SPLINE
SPL {X  -154.923, Y  +342.556, Z    +0.000, E1   +23.930, E3 +323700.309}
SPL {X  -158.138, Y  +358.230, Z    +0.000, E1   +16.243, E3 +323709.267}
SPL {X  -159.407, Y  +368.849, Z    +0.000, E1   +10.504, E3 +323712.867}
SPL {X  -159.931, Y  +378.162, Z    +0.000, E1    +5.020, E3 +323714.852}
SPL {X  -159.990, Y  +384.616, Z    +0.000, E1    +0.627, E3 +323715.691}
SPL {X  -159.990, Y  +387.962, Z    +0.000, E1    -2.241, E3 +323716.048}
SPL {X  -159.990, Y  +390.921, Z    +0.000, E1    -5.111, E3 +323716.413}
SPL {X  -159.990, Y  +395.719, Z    +0.000, E1   -10.396, E3 +323717.232}
SPL {X  -159.990, Y  +400.739, Z    +0.000, E1   -16.236, E3 +323718.430}
SPL {X  -159.990, Y  +409.482, Z    +0.000, E1   -25.418, E3 +323721.635}
SPL {X  -159.990, Y  +440.741, Z    +0.000, E1   -43.570, E3 +323742.292}
SPL {X  -159.990, Y  +488.072, Z    +0.000, E1   -48.834, E3 +323803.414}
SPL {X  -159.990, Y  +495.397, Z    +0.000, E1   -48.860, E3 +323816.963}
SPL {X  -159.990, Y  +502.531, Z    +0.000, E1   -48.834, E3 +323830.242}
SPL {X  -159.990, Y  +508.013, Z    +0.000, E1   -48.835, E3 +323840.377}
SPL {X  -159.990, Y  +513.813, Z    +0.000, E1   -48.843, E3 +323851.125}
SPL {X  -159.990, Y  +522.177, Z    +0.000, E1   -48.881, E3 +323866.602}
SPL {X  -159.990, Y  +532.076, Z    +0.000, E1   -48.872, E3 +323884.975}
SPL {X  -159.990, Y  +539.248, Z    +0.000, E1   -48.832, E3 +323898.343}
SPL {X  -159.990, Y  +544.926, Z    +0.000, E1   -48.835, E3 +323908.872}
SPL {X  -159.990, Y  +550.252, Z    +0.000, E1   -48.827, E3 +323918.778}
SPL {X  -159.990, Y  +555.692, Z    +0.000, E1   -48.830, E3 +323928.875}
SPL {X  -159.990, Y  +561.308, Z    +0.000, E1   -48.827, E3 +323939.322}
SPL {X  -159.990, Y  +566.669, Z    +0.000, E1   -48.820, E3 +323949.271}
SPL {X  -159.990, Y  +572.248, Z    +0.000, E1   -48.830, E3 +323959.616}
SPL {X  -159.990, Y  +577.770, Z    +0.000, E1   -48.821, E3 +323969.863}
SPL {X  -159.990, Y  +583.108, Z    +0.000, E1   -48.828, E3 +323979.765}
SPL {X  -159.990, Y  +588.804, Z    +0.000, E1   -48.829, E3 +323990.322}
SPL {X  -159.990, Y  +594.280, Z    +0.000, E1   -48.826, E3 +324000.484}
SPL {X  -159.990, Y  +600.107, Z    +0.000, E1   -48.833, E3 +324011.298}
SPL {X  -159.990, Y  +605.910, Z    +0.000, E1   -48.823, E3 +324022.077}
SPL {X  -159.990, Y  +611.566, Z    +0.000, E1   -48.829, E3 +324032.566}
SPL {X  -159.990, Y  +617.357, Z    +0.000, E1   -48.824, E3 +324043.321}
SPL {X  -159.990, Y  +622.965, Z    +0.000, E1   -48.826, E3 +324053.720}
SPL {X  -159.990, Y  +629.255, Z    +0.000, E1   -48.834, E3 +324065.387}
SPL {X  -159.990, Y  +634.905, Z    +0.000, E1   -48.821, E3 +324075.884}
SPL {X  -159.990, Y  +640.372, Z    +0.000, E1   -48.828, E3 +324086.021}
SPL {X  -159.990, Y  +646.939, Z    +0.000, E1   -48.838, E3 +324098.191}
SPL {X  -159.990, Y  +653.448, Z    +0.000, E1   -48.827, E3 +324110.286}
SPL {X  -159.990, Y  +659.039, Z    +0.000, E1   -48.826, E3 +324120.650}
SPL {X  -159.990, Y  +664.817, Z    +0.000, E1   -48.832, E3 +324131.365}
SPL {X  -159.990, Y  +671.221, Z    +0.000, E1   -48.836, E3 +324143.238}
SPL {X  -159.887, Y  +677.230, Z    +0.000, E1   -48.811, E3 +324154.504}
SPL {X  -159.602, Y  +682.629, Z    +0.000, E1   -48.761, E3 +324164.837}
SPL {X  -159.150, Y  +687.876, Z    +0.000, E1   -48.673, E3 +324175.076}
SPL {X  -158.569, Y  +692.776, Z    +0.000, E1   -48.570, E3 +324184.784}
SPL {X  -157.870, Y  +697.458, Z    +0.000, E1   -48.439, E3 +324194.213}
SPL {X  -157.028, Y  +702.144, Z    +0.000, E1   -48.297, E3 +324203.761}
SPL {X  -155.977, Y  +707.110, Z    +0.000, E1   -48.106, E3 +324214.065}
SPL {X  -154.657, Y  +712.464, Z    +0.000, E1   -47.874, E3 +324225.349}
SPL {X  -153.406, Y  +716.924, Z    +0.000, E1   -47.628, E3 +324234.915}
SPL {X  -152.020, Y  +721.367, Z    +0.000, E1   -47.374, E3 +324244.566}
SPL {X  -150.440, Y  +725.947, Z    +0.000, E1   -47.070, E3 +324254.671}
SPL {X  -148.730, Y  +730.459, Z    +0.000, E1   -46.749, E3 +324264.722}
SPL {X  -147.178, Y  +734.233, Z    +0.000, E1   -46.439, E3 +324273.256}
SPL {X  -140.263, Y  +748.461, Z    +0.000, E1   -42.675, E3 +324331.594}
ENDSPLINE

SPLINE
SPL {X  -141.835, Y  +745.525, Z    +0.000, E1   -39.068, E3 +324363.595}
SPL {X  -152.406, Y  +720.176, Z    +0.000, E1   -27.814, E3 +324414.808}
SPL {X  -158.165, Y  +695.595, Z    +0.000, E1   -16.189, E3 +324430.706}
SPL {X  -159.572, Y  +683.063, Z    +0.000, E1    -9.282, E3 +324434.713}
SPL {X  -159.928, Y  +675.946, Z    +0.000, E1    -5.007, E3 +324436.134}
SPL {X  -159.990, Y  +671.468, Z    +0.000, E1    -2.030, E3 +324436.730}
SPL {X  -159.990, Y  +667.678, Z    +0.000, E1    +0.783, E3 +324437.080}
SPL {X  -159.990, Y  +663.139, Z    +0.000, E1    +5.135, E3 +324437.597}
SPL {X  -159.990, Y  +658.551, Z    +0.000, E1   +10.313, E3 +324438.371}
SPL {X  -159.990, Y  +653.526, Z    +0.000, E1   +16.156, E3 +324439.606}
SPL {X  -159.990, Y  +644.434, Z    +0.000, E1   +25.921, E3 +324442.801}
SPL {X  -159.990, Y  +612.255, Z    +0.000, E1   +44.102, E3 +324464.682}
SPL {X  -159.990, Y  +562.879, Z    +0.000, E1   +49.634, E3 +324526.271}
SPL {X  -159.990, Y  +554.544, Z    +0.000, E1   +49.649, E3 +324541.296}
SPL {X  -159.990, Y  +547.278, Z    +0.000, E1   +49.619, E3 +324554.455}
SPL {X  -159.990, Y  +540.489, Z    +0.000, E1   +49.634, E3 +324566.681}
SPL {X  -159.990, Y  +530.983, Z    +0.000, E1   +49.676, E3 +324583.752}
SPL {X  -159.990, Y  +522.804, Z    +0.000, E1   +49.620, E3 +324598.592}
SPL {X  -159.990, Y  +515.173, Z    +0.000, E1   +49.653, E3 +324612.330}
SPL {X  -159.990, Y  +505.472, Z    +0.000, E1   +49.465, E3 +324631.135}
ENDSPLINE

SPLINE
SPL {X  -159.990, Y  +518.841, Z    +0.000, E1   +41.643, E3 +324649.543}
ENDSPLINE

SPLINE
SPL {X  -159.990, Y  +508.096, Z    +0.000, E1   +42.952, E3 +324666.810}
SPL {X  -159.990, Y  +500.642, Z    +0.000, E1   +43.747, E3 +324678.731}
SPL {X  -159.990, Y  +495.820, Z    +0.000, E1   +44.207, E3 +324686.618}
SPL {X  -159.990, Y  +487.435, Z    +0.000, E1   +45.185, E3 +324698.910}
SPL {X  -159.990, Y  +477.648, Z    +0.000, E1   +46.080, E3 +324713.907}
SPL {X  -159.990, Y  +469.952, Z    +0.000, E1   +46.750, E3 +324725.415}
SPL {X  -159.990, Y  +460.762, Z    +0.000, E1   +47.755, E3 +324737.551}
SPL {X  -159.990, Y  +451.028, Z    +0.000, E1   +48.723, E3 +324750.163}
SPL {X  -159.990, Y  +441.023, Z    +0.000, E1   +49.655, E3 +324762.997}
SPL {X  -159.990, Y  +431.096, Z    +0.000, E1   +50.075, E3 +324778.285}
SPL {X  -159.990, Y  +423.834, Z    +0.000, E1   +50.037, E3 +324791.258}
SPL {X  -159.990, Y  +417.693, Z    +0.000, E1   +50.049, E3 +324802.156}
SPL {X  -159.990, Y  +411.447, Z    +0.000, E1   +50.039, E3 +324813.275}
SPL {X  -159.990, Y  +406.170, Z    +0.000, E1   +50.036, E3 +324822.647}
SPL {X  -159.990, Y  +399.787, Z    +0.000, E1   +50.064, E3 +324833.955}
SPL {X  -159.990, Y  +393.038, Z    +0.000, E1   +50.038, E3 +324845.989}
SPL {X  -159.990, Y  +387.356, Z    +0.000, E1   +50.042, E3 +324856.100}
SPL {X  -159.956, Y  +379.183, Z    +0.000, E1   +50.071, E3 +324870.614}
SPL {X  -159.413, Y  +368.921, Z    +0.000, E1   +49.998, E3 +324889.389}
SPL {X  -158.412, Y  +360.086, Z    +0.000, E1   +49.787, E3 +324906.191}
SPL {X  -157.077, Y  +352.107, Z    +0.000, E1   +49.567, E3 +324921.742}
SPL {X  -155.744, Y  +345.884, Z    +0.000, E1   +49.283, E3 +324934.229}
SPL {X  -154.686, Y  +341.646, Z    +0.000, E1   +49.094, E3 +324942.855}
SPL {X  -153.089, Y  +336.017, Z    +0.000, E1   +48.817, E3 +324954.464}
SPL {X  -151.481, Y  +331.019, Z    +0.000, E1   +48.491, E3 +324965.012}
SPL {X  -149.787, Y  +326.281, Z    +0.000, E1   +48.192, E3 +324975.100}
SPL {X  -148.124, Y  +322.035, Z    +0.000, E1   +47.846, E3 +324984.324}
SPL {X  -146.510, Y  +318.222, Z    +0.000, E1   +47.558, E3 +324992.636}
SPL {X  -141.189, Y  +307.250, Z    +0.000, E1   +40.067, E3 +325078.810}
ENDSPLINE

SPLINE
SPL {X  -154.923, Y  +342.556, Z    +0.000, E1   +23.930, E3 +325140.309}
SPL {X  -158.138, Y  +358.230, Z    +0.000, E1   +16.243, E3 +325149.267}
SPL {X  -159.647, Y  +372.034, Z    +0.000, E1    +8.739, E3 +325153.631}
SPL {X  -159.989, Y  +381.927, Z    +0.000, E1    +2.565, E3 +325155.391}
SPL {X  -159.990, Y  +386.909, Z    +0.000, E1    -1.211, E3 +325155.934}
SPL {X  -159.990, Y  +390.921, Z    +0.000, E1    -5.111, E3 +325156.413}
SPL {X  -159.990, Y  +395.719, Z    +0.000, E1   -10.396, E3 +325157.232}
SPL {X  -159.990, Y  +400.739, Z    +0.000, E1   -16.236, E3 +325158.430}
SPL {X  -159.990, Y  +409.482, Z    +0.000, E1   -25.418, E3 +325161.635}
SPL {X  -159.990, Y  +440.741, Z    +0.000, E1   -43.570, E3 +325182.292}
SPL {X  -159.990, Y  +488.072, Z    +0.000, E1   -48.834, E3 +325243.414}
SPL {X  -159.990, Y  +495.397, Z    +0.000, E1   -48.860, E3 +325256.963}
SPL {X  -159.990, Y  +502.531, Z    +0.000, E1   -48.834, E3 +325270.242}
SPL {X  -159.990, Y  +508.013, Z    +0.000, E1   -48.835, E3 +325280.377}
SPL {X  -159.990, Y  +513.813, Z    +0.000, E1   -48.843, E3 +325291.125}
SPL {X  -159.990, Y  +519.614, Z    +0.000, E1   -48.832, E3 +325301.926}
SPL {X  -159.990, Y  +527.523, Z    +0.000, E1   -48.881, E3 +325316.507}
SPL {X  -159.990, Y  +537.185, Z    +0.000, E1   -48.874, E3 +325334.454}
SPL {X  -159.990, Y  +544.926, Z    +0.000, E1   -48.835, E3 +325348.872}
SPL {X  -159.990, Y  +550.252, Z    +0.000, E1   -48.827, E3 +325358.778}
SPL {X  -159.990, Y  +555.692, Z    +0.000, E1   -48.830, E3 +325368.875}
SPL {X  -159.990, Y  +561.308, Z    +0.000, E1   -48.827, E3 +325379.322}
SPL {X  -159.990, Y  +566.669, Z    +0.000, E1   -48.820, E3 +325389.271}
SPL {X  -159.990, Y  +572.248, Z    +0.000, E1   -48.830, E3 +325399.616}
SPL {X  -159.990, Y  +577.770, Z    +0.000, E1   -48.821, E3 +325409.863}
SPL {X  -159.990, Y  +583.108, Z    +0.000, E1   -48.828, E3 +325419.765}
SPL {X  -159.990, Y  +588.804, Z    +0.000, E1   -48.829, E3 +325430.322}
SPL {X  -159.990, Y  +594.280, Z    +0.000, E1   -48.826, E3 +325440.484}
SPL {X  -159.990, Y  +600.107, Z    +0.000, E1   -48.833, E3 +325451.298}
SPL {X  -159.990, Y  +605.910, Z    +0.000, E1   -48.823, E3 +325462.077}
SPL {X  -159.990, Y  +611.566, Z    +0.000, E1   -48.829, E3 +325472.566}
SPL {X  -159.990, Y  +617.357, Z    +0.000, E1   -48.824, E3 +325483.321}
SPL {X  -159.990, Y  +622.965, Z    +0.000, E1   -48.826, E3 +325493.720}
SPL {X  -159.990, Y  +629.255, Z    +0.000, E1   -48.834, E3 +325505.387}
SPL {X  -159.990, Y  +634.905, Z    +0.000, E1   -48.821, E3 +325515.884}
SPL {X  -159.990, Y  +640.372, Z    +0.000, E1   -48.828, E3 +325526.021}
SPL {X  -159.990, Y  +646.939, Z    +0.000, E1   -48.838, E3 +325538.191}
SPL {X  -159.990, Y  +653.448, Z    +0.000, E1   -48.827, E3 +325550.286}
SPL {X  -159.990, Y  +659.039, Z    +0.000, E1   -48.826, E3 +325560.650}
SPL {X  -159.990, Y  +664.817, Z    +0.000, E1   -48.832, E3 +325571.365}
SPL {X  -159.990, Y  +671.221, Z    +0.000, E1   -48.836, E3 +325583.238}
SPL {X  -159.887, Y  +677.230, Z    +0.000, E1   -48.811, E3 +325594.504}
SPL {X  -159.602, Y  +682.629, Z    +0.000, E1   -48.761, E3 +325604.837}
SPL {X  -159.150, Y  +687.876, Z    +0.000, E1   -48.673, E3 +325615.076}
SPL {X  -158.569, Y  +692.776, Z    +0.000, E1   -48.570, E3 +325624.784}
SPL {X  -157.870, Y  +697.458, Z    +0.000, E1   -48.439, E3 +325634.213}
SPL {X  -157.028, Y  +702.144, Z    +0.000, E1   -48.297, E3 +325643.761}
SPL {X  -155.977, Y  +707.110, Z    +0.000, E1   -48.106, E3 +325654.065}
SPL {X  -154.657, Y  +712.464, Z    +0.000, E1   -47.874, E3 +325665.349}
SPL {X  -153.406, Y  +716.924, Z    +0.000, E1   -47.628, E3 +325674.915}
SPL {X  -152.020, Y  +721.367, Z    +0.000, E1   -47.374, E3 +325684.566}
SPL {X  -150.440, Y  +725.947, Z    +0.000, E1   -47.070, E3 +325694.671}
SPL {X  -148.730, Y  +730.459, Z    +0.000, E1   -46.749, E3 +325704.722}
SPL {X  -147.178, Y  +734.233, Z    +0.000, E1   -46.439, E3 +325713.256}
SPL {X  -140.263, Y  +748.461, Z    +0.000, E1   -42.675, E3 +325771.594}
ENDSPLINE

SPLINE
SPL {X  -141.835, Y  +745.525, Z    +0.000, E1   -39.068, E3 +325803.595}
SPL {X  -152.406, Y  +720.176, Z    +0.000, E1   -27.814, E3 +325854.808}
SPL {X  -158.165, Y  +695.595, Z    +0.000, E1   -16.189, E3 +325870.706}
SPL {X  -159.572, Y  +683.063, Z    +0.000, E1    -9.282, E3 +325874.713}
SPL {X  -159.928, Y  +675.946, Z    +0.000, E1    -5.007, E3 +325876.134}
SPL {X  -159.990, Y  +671.468, Z    +0.000, E1    -2.030, E3 +325876.730}
SPL {X  -159.990, Y  +667.678, Z    +0.000, E1    +0.783, E3 +325877.080}
SPL {X  -159.990, Y  +663.139, Z    +0.000, E1    +5.135, E3 +325877.597}
SPL {X  -159.990, Y  +658.551, Z    +0.000, E1   +10.313, E3 +325878.371}
SPL {X  -159.990, Y  +653.526, Z    +0.000, E1   +16.156, E3 +325879.606}
SPL {X  -159.990, Y  +644.434, Z    +0.000, E1   +25.921, E3 +325882.801}
SPL {X  -159.990, Y  +612.255, Z    +0.000, E1   +44.102, E3 +325904.682}
SPL {X  -159.990, Y  +562.879, Z    +0.000, E1   +49.634, E3 +325966.271}
SPL {X  -159.990, Y  +554.544, Z    +0.000, E1   +49.649, E3 +325981.296}
SPL {X  -159.990, Y  +547.278, Z    +0.000, E1   +49.619, E3 +325994.455}
SPL {X  -159.990, Y  +540.489, Z    +0.000, E1   +49.634, E3 +326006.681}
SPL {X  -159.990, Y  +530.983, Z    +0.000, E1   +49.676, E3 +326023.752}
SPL {X  -159.990, Y  +522.804, Z    +0.000, E1   +49.620, E3 +326038.592}
SPL {X  -159.990, Y  +515.173, Z    +0.000, E1   +49.653, E3 +326052.330}
SPL {X  -159.990, Y  +505.472, Z    +0.000, E1   +49.465, E3 +326071.135}
ENDSPLINE

SPLINE
SPL {X  -159.990, Y  +520.622, Z    +0.000, E1   +41.395, E3 +326086.672}
ENDSPLINE

SPLINE
SPL {X  -159.990, Y  +512.735, Z    +0.000, E1   +42.369, E3 +326099.523}
SPL {X  -159.990, Y  +505.924, Z    +0.000, E1   +43.199, E3 +326110.181}
SPL {X  -159.990, Y  +497.983, Z    +0.000, E1   +44.027, E3 +326123.054}
SPL {X  -159.990, Y  +489.703, Z    +0.000, E1   +44.938, E3 +326135.473}
SPL {X  -159.990, Y  +482.131, Z    +0.000, E1   +45.680, E3 +326147.053}
SPL {X  -159.990, Y  +472.111, Z    +0.000, E1   +46.581, E3 +326162.185}
SPL {X  -159.990, Y  +462.892, Z    +0.000, E1   +47.497, E3 +326174.899}
SPL {X  -159.990, Y  +450.424, Z    +0.000, E1   +48.824, E3 +326190.863}
SPL {X  -159.990, Y  +436.919, Z    +0.000, E1   +49.944, E3 +326208.632}
SPL {X  -159.990, Y  +429.517, Z    +0.000, E1   +50.043, E3 +326221.146}
SPL {X  -159.990, Y  +423.834, Z    +0.000, E1   +50.037, E3 +326231.258}
SPL {X  -159.990, Y  +417.693, Z    +0.000, E1   +50.049, E3 +326242.156}
SPL {X  -159.990, Y  +411.447, Z    +0.000, E1   +50.039, E3 +326253.275}
SPL {X  -159.990, Y  +403.654, Z    +0.000, E1   +50.076, E3 +326267.065}
SPL {X  -159.990, Y  +394.612, Z    +0.000, E1   +50.064, E3 +326283.153}
SPL {X  -159.990, Y  +387.356, Z    +0.000, E1   +50.042, E3 +326296.100}
SPL {X  -159.956, Y  +379.183, Z    +0.000, E1   +50.071, E3 +326310.614}
SPL {X  -159.413, Y  +368.921, Z    +0.000, E1   +49.998, E3 +326329.389}
SPL {X  -158.412, Y  +360.086, Z    +0.000, E1   +49.787, E3 +326346.191}
SPL {X  -157.077, Y  +352.107, Z    +0.000, E1   +49.567, E3 +326361.742}
SPL {X  -155.744, Y  +345.884, Z    +0.000, E1   +49.283, E3 +326374.229}
SPL {X  -154.686, Y  +341.646, Z    +0.000, E1   +49.094, E3 +326382.855}
SPL {X  -153.089, Y  +336.017, Z    +0.000, E1   +48.817, E3 +326394.464}
SPL {X  -151.481, Y  +331.019, Z    +0.000, E1   +48.491, E3 +326405.012}
SPL {X  -150.221, Y  +327.451, Z    +0.000, E1   +48.251, E3 +326412.616}
SPL {X  -148.587, Y  +323.181, Z    +0.000, E1   +47.960, E3 +326421.800}
SPL {X  -146.510, Y  +318.222, Z    +0.000, E1   +47.558, E3 +326432.636}
SPL {X  -141.189, Y  +307.250, Z    +0.000, E1   +40.067, E3 +326518.810}
ENDSPLINE

SPLINE
SPL {X  -154.923, Y  +342.556, Z    +0.000, E1   +23.930, E3 +326580.309}
SPL {X  -158.138, Y  +358.230, Z    +0.000, E1   +16.243, E3 +326589.267}
SPL {X  -159.407, Y  +368.849, Z    +0.000, E1   +10.504, E3 +326592.867}
SPL {X  -159.931, Y  +378.162, Z    +0.000, E1    +5.020, E3 +326594.852}
SPL {X  -159.990, Y  +383.297, Z    +0.000, E1    +1.526, E3 +326595.557}
SPL {X  -159.990, Y  +386.909, Z    +0.000, E1    -1.211, E3 +326595.934}
SPL {X  -159.990, Y  +390.921, Z    +0.000, E1    -5.111, E3 +326596.413}
SPL {X  -159.990, Y  +395.719, Z    +0.000, E1   -10.396, E3 +326597.232}
SPL {X  -159.990, Y  +400.739, Z    +0.000, E1   -16.236, E3 +326598.430}
SPL {X  -159.990, Y  +407.669, Z    +0.000, E1   -23.731, E3 +326600.753}
SPL {X  -159.990, Y  +417.102, Z    +0.000, E1   -32.094, E3 +326605.313}
SPL {X  -159.990, Y  +440.741, Z    +0.000, E1   -43.570, E3 +326622.292}
SPL {X  -159.990, Y  +488.072, Z    +0.000, E1   -48.834, E3 +326683.414}
SPL {X  -159.990, Y  +495.397, Z    +0.000, E1   -48.860, E3 +326696.963}
SPL {X  -159.990, Y  +502.531, Z    +0.000, E1   -48.834, E3 +326710.242}
SPL {X  -159.990, Y  +508.013, Z    +0.000, E1   -48.835, E3 +326720.377}
SPL {X  -159.990, Y  +513.813, Z    +0.000, E1   -48.843, E3 +326731.125}
SPL {X  -159.990, Y  +522.177, Z    +0.000, E1   -48.881, E3 +326746.602}
SPL {X  -159.990, Y  +532.076, Z    +0.000, E1   -48.872, E3 +326764.975}
SPL {X  -159.990, Y  +539.248, Z    +0.000, E1   -48.832, E3 +326778.343}
SPL {X  -159.990, Y  +544.926, Z    +0.000, E1   -48.835, E3 +326788.872}
SPL {X  -159.990, Y  +550.252, Z    +0.000, E1   -48.827, E3 +326798.778}
SPL {X  -159.990, Y  +555.692, Z    +0.000, E1   -48.830, E3 +326808.875}
SPL {X  -159.990, Y  +561.308, Z    +0.000, E1   -48.827, E3 +326819.322}
SPL {X  -159.990, Y  +566.669, Z    +0.000, E1   -48.820, E3 +326829.271}
SPL {X  -159.990, Y  +572.248, Z    +0.000, E1   -48.830, E3 +326839.616}
SPL {X  -159.990, Y  +577.770, Z    +0.000, E1   -48.821, E3 +326849.863}
SPL {X  -159.990, Y  +583.108, Z    +0.000, E1   -48.828, E3 +326859.765}
SPL {X  -159.990, Y  +588.804, Z    +0.000, E1   -48.829, E3 +326870.322}
SPL {X  -159.990, Y  +594.280, Z    +0.000, E1   -48.826, E3 +326880.484}
SPL {X  -159.990, Y  +600.107, Z    +0.000, E1   -48.833, E3 +326891.298}
SPL {X  -159.990, Y  +605.910, Z    +0.000, E1   -48.823, E3 +326902.077}
SPL {X  -159.990, Y  +611.566, Z    +0.000, E1   -48.829, E3 +326912.566}
SPL {X  -159.990, Y  +617.357, Z    +0.000, E1   -48.824, E3 +326923.321}
SPL {X  -159.990, Y  +622.965, Z    +0.000, E1   -48.826, E3 +326933.720}
SPL {X  -159.990, Y  +629.255, Z    +0.000, E1   -48.834, E3 +326945.387}
SPL {X  -159.990, Y  +634.905, Z    +0.000, E1   -48.821, E3 +326955.884}
SPL {X  -159.990, Y  +640.372, Z    +0.000, E1   -48.828, E3 +326966.021}
SPL {X  -159.990, Y  +646.939, Z    +0.000, E1   -48.838, E3 +326978.191}
SPL {X  -159.990, Y  +653.448, Z    +0.000, E1   -48.827, E3 +326990.286}
SPL {X  -159.990, Y  +659.039, Z    +0.000, E1   -48.826, E3 +327000.650}
SPL {X  -159.990, Y  +664.817, Z    +0.000, E1   -48.832, E3 +327011.365}
SPL {X  -159.990, Y  +671.221, Z    +0.000, E1   -48.836, E3 +327023.238}
SPL {X  -159.887, Y  +677.230, Z    +0.000, E1   -48.811, E3 +327034.504}
SPL {X  -159.602, Y  +682.629, Z    +0.000, E1   -48.761, E3 +327044.837}
SPL {X  -159.150, Y  +687.876, Z    +0.000, E1   -48.673, E3 +327055.076}
SPL {X  -158.569, Y  +692.776, Z    +0.000, E1   -48.570, E3 +327064.784}
SPL {X  -157.870, Y  +697.458, Z    +0.000, E1   -48.439, E3 +327074.213}
SPL {X  -157.028, Y  +702.144, Z    +0.000, E1   -48.297, E3 +327083.761}
SPL {X  -155.977, Y  +707.110, Z    +0.000, E1   -48.106, E3 +327094.065}
SPL {X  -154.657, Y  +712.464, Z    +0.000, E1   -47.874, E3 +327105.349}
SPL {X  -153.406, Y  +716.924, Z    +0.000, E1   -47.628, E3 +327114.915}
SPL {X  -152.020, Y  +721.367, Z    +0.000, E1   -47.374, E3 +327124.566}
SPL {X  -150.440, Y  +725.947, Z    +0.000, E1   -47.070, E3 +327134.671}
SPL {X  -148.730, Y  +730.459, Z    +0.000, E1   -46.749, E3 +327144.722}
SPL {X  -147.178, Y  +734.233, Z    +0.000, E1   -46.439, E3 +327153.256}
SPL {X  -140.263, Y  +748.461, Z    +0.000, E1   -42.675, E3 +327211.594}
ENDSPLINE

SPLINE
SPL {X  -141.835, Y  +745.525, Z    +0.000, E1   -39.068, E3 +327243.595}
SPL {X  -152.406, Y  +720.176, Z    +0.000, E1   -27.814, E3 +327294.808}
SPL {X  -157.542, Y  +699.382, Z    +0.000, E1   -18.086, E3 +327309.141}
SPL {X  -159.386, Y  +685.393, Z    +0.000, E1   -10.664, E3 +327314.095}
SPL {X  -159.928, Y  +675.946, Z    +0.000, E1    -5.007, E3 +327316.134}
SPL {X  -159.990, Y  +671.468, Z    +0.000, E1    -2.030, E3 +327316.730}
SPL {X  -159.990, Y  +667.678, Z    +0.000, E1    +0.783, E3 +327317.080}
SPL {X  -159.990, Y  +663.139, Z    +0.000, E1    +5.135, E3 +327317.597}
SPL {X  -159.990, Y  +658.551, Z    +0.000, E1   +10.313, E3 +327318.371}
SPL {X  -159.990, Y  +653.526, Z    +0.000, E1   +16.156, E3 +327319.606}
SPL {X  -159.990, Y  +644.434, Z    +0.000, E1   +25.921, E3 +327322.801}
SPL {X  -159.990, Y  +612.255, Z    +0.000, E1   +44.102, E3 +327344.682}
SPL {X  -159.990, Y  +561.053, Z    +0.000, E1   +49.668, E3 +327409.515}
SPL {X  -159.990, Y  +552.984, Z    +0.000, E1   +49.619, E3 +327424.156}
SPL {X  -159.990, Y  +547.278, Z    +0.000, E1   +49.619, E3 +327434.455}
SPL {X  -159.990, Y  +538.738, Z    +0.000, E1   +49.672, E3 +327449.779}
SPL {X  -159.990, Y  +529.436, Z    +0.000, E1   +49.638, E3 +327466.603}
SPL {X  -159.990, Y  +520.280, Z    +0.000, E1   +49.665, E3 +327483.082}
SPL {X  -159.990, Y  +511.038, Z    +0.000, E1   +49.636, E3 +327499.832}
SPL {X  -159.990, Y  +504.260, Z    +0.000, E1   +49.614, E3 +327512.105}
SPL {X  -159.990, Y  +503.881, Z    +0.000, E1   +48.376, E3 +327520.092}
ENDSPLINE

SPLINE
SPL {X  -159.990, Y  +520.622, Z    +0.000, E1   +41.395, E3 +327526.672}
ENDSPLINE

SPLINE
SPL {X  -159.990, Y  +512.735, Z    +0.000, E1   +42.369, E3 +327539.523}
SPL {X  -159.990, Y  +505.924, Z    +0.000, E1   +43.199, E3 +327550.181}
SPL {X  -159.990, Y  +497.983, Z    +0.000, E1   +44.027, E3 +327563.054}
SPL {X  -159.990, Y  +489.703, Z    +0.000, E1   +44.938, E3 +327575.473}
SPL {X  -159.990, Y  +484.712, Z    +0.000, E1   +45.426, E3 +327583.087}
SPL {X  -159.990, Y  +477.648, Z    +0.000, E1   +46.080, E3 +327593.907}
SPL {X  -159.990, Y  +469.952, Z    +0.000, E1   +46.750, E3 +327605.415}
SPL {X  -159.990, Y  +462.892, Z    +0.000, E1   +47.497, E3 +327614.899}
SPL {X  -159.990, Y  +450.424, Z    +0.000, E1   +48.824, E3 +327630.863}
SPL {X  -159.990, Y  +436.919, Z    +0.000, E1   +49.944, E3 +327648.632}
SPL {X  -159.990, Y  +429.517, Z    +0.000, E1   +50.043, E3 +327661.146}
SPL {X  -159.990, Y  +423.834, Z    +0.000, E1   +50.037, E3 +327671.258}
SPL {X  -159.990, Y  +417.693, Z    +0.000, E1   +50.049, E3 +327682.156}
SPL {X  -159.990, Y  +408.922, Z    +0.000, E1   +50.085, E3 +327697.686}
SPL {X  -159.990, Y  +399.787, Z    +0.000, E1   +50.064, E3 +327713.955}
SPL {X  -159.990, Y  +393.038, Z    +0.000, E1   +50.038, E3 +327725.989}
SPL {X  -159.990, Y  +385.182, Z    +0.000, E1   +50.081, E3 +327739.906}
SPL {X  -159.906, Y  +377.302, Z    +0.000, E1   +50.024, E3 +327754.067}
SPL {X  -159.545, Y  +370.569, Z    +0.000, E1   +49.982, E3 +327766.380}
SPL {X  -158.871, Y  +363.614, Z    +0.000, E1   +49.855, E3 +327779.459}
SPL {X  -158.179, Y  +358.495, Z    +0.000, E1   +49.715, E3 +327789.308}
SPL {X  -157.354, Y  +353.576, Z    +0.000, E1   +49.583, E3 +327798.894}
SPL {X  -156.029, Y  +347.121, Z    +0.000, E1   +49.358, E3 +327811.711}
SPL {X  -154.686, Y  +341.646, Z    +0.000, E1   +49.094, E3 +327822.855}
SPL {X  -153.089, Y  +336.017, Z    +0.000, E1   +48.817, E3 +327834.464}
SPL {X  -151.481, Y  +331.019, Z    +0.000, E1   +48.491, E3 +327845.012}
SPL {X  -149.787, Y  +326.281, Z    +0.000, E1   +48.192, E3 +327855.100}
SPL {X  -148.124, Y  +322.035, Z    +0.000, E1   +47.846, E3 +327864.324}
SPL {X  -146.510, Y  +318.222, Z    +0.000, E1   +47.558, E3 +327872.636}
SPL {X  -141.189, Y  +307.250, Z    +0.000, E1   +40.067, E3 +327958.810}
ENDSPLINE

SPLINE
SPL {X  -154.923, Y  +342.556, Z    +0.000, E1   +23.930, E3 +328020.309}
SPL {X  -158.138, Y  +358.230, Z    +0.000, E1   +16.243, E3 +328029.267}
SPL {X  -159.647, Y  +372.034, Z    +0.000, E1    +8.739, E3 +328033.631}
SPL {X  -159.989, Y  +381.927, Z    +0.000, E1    +2.565, E3 +328035.391}
SPL {X  -159.990, Y  +386.909, Z    +0.000, E1    -1.211, E3 +328035.934}
SPL {X  -159.990, Y  +390.921, Z    +0.000, E1    -5.111, E3 +328036.413}
SPL {X  -159.990, Y  +395.719, Z    +0.000, E1   -10.396, E3 +328037.232}
SPL {X  -159.990, Y  +400.739, Z    +0.000, E1   -16.236, E3 +328038.430}
SPL {X  -159.990, Y  +409.482, Z    +0.000, E1   -25.418, E3 +328041.635}
SPL {X  -159.990, Y  +440.741, Z    +0.000, E1   -43.570, E3 +328062.292}
SPL {X  -159.990, Y  +489.732, Z    +0.000, E1   -48.863, E3 +328126.450}
SPL {X  -159.990, Y  +496.901, Z    +0.000, E1   -48.832, E3 +328139.797}
SPL {X  -159.990, Y  +502.531, Z    +0.000, E1   -48.834, E3 +328150.242}
SPL {X  -159.990, Y  +508.013, Z    +0.000, E1   -48.835, E3 +328160.377}
SPL {X  -159.990, Y  +513.813, Z    +0.000, E1   -48.843, E3 +328171.125}
SPL {X  -159.990, Y  +522.177, Z    +0.000, E1   -48.881, E3 +328186.602}
SPL {X  -159.990, Y  +532.076, Z    +0.000, E1   -48.872, E3 +328204.975}
SPL {X  -159.990, Y  +539.248, Z    +0.000, E1   -48.832, E3 +328218.343}
SPL {X  -159.990, Y  +544.926, Z    +0.000, E1   -48.835, E3 +328228.872}
SPL {X  -159.990, Y  +550.252, Z    +0.000, E1   -48.827, E3 +328238.778}
SPL {X  -159.990, Y  +555.692, Z    +0.000, E1   -48.830, E3 +328248.875}
SPL {X  -159.990, Y  +561.308, Z    +0.000, E1   -48.827, E3 +328259.322}
SPL {X  -159.990, Y  +566.669, Z    +0.000, E1   -48.820, E3 +328269.271}
SPL {X  -159.990, Y  +572.248, Z    +0.000, E1   -48.830, E3 +328279.616}
SPL {X  -159.990, Y  +577.770, Z    +0.000, E1   -48.821, E3 +328289.863}
SPL {X  -159.990, Y  +583.108, Z    +0.000, E1   -48.828, E3 +328299.765}
SPL {X  -159.990, Y  +588.804, Z    +0.000, E1   -48.829, E3 +328310.322}
SPL {X  -159.990, Y  +594.280, Z    +0.000, E1   -48.826, E3 +328320.484}
SPL {X  -159.990, Y  +600.107, Z    +0.000, E1   -48.833, E3 +328331.298}
SPL {X  -159.990, Y  +605.910, Z    +0.000, E1   -48.823, E3 +328342.077}
SPL {X  -159.990, Y  +611.566, Z    +0.000, E1   -48.829, E3 +328352.566}
SPL {X  -159.990, Y  +617.357, Z    +0.000, E1   -48.824, E3 +328363.321}
SPL {X  -159.990, Y  +622.965, Z    +0.000, E1   -48.826, E3 +328373.720}
SPL {X  -159.990, Y  +629.255, Z    +0.000, E1   -48.834, E3 +328385.387}
SPL {X  -159.990, Y  +634.905, Z    +0.000, E1   -48.821, E3 +328395.884}
SPL {X  -159.990, Y  +640.372, Z    +0.000, E1   -48.828, E3 +328406.021}
SPL {X  -159.990, Y  +646.939, Z    +0.000, E1   -48.838, E3 +328418.191}
SPL {X  -159.990, Y  +653.448, Z    +0.000, E1   -48.827, E3 +328430.286}
SPL {X  -159.990, Y  +659.039, Z    +0.000, E1   -48.826, E3 +328440.650}
SPL {X  -159.990, Y  +664.817, Z    +0.000, E1   -48.832, E3 +328451.365}
SPL {X  -159.990, Y  +671.221, Z    +0.000, E1   -48.836, E3 +328463.238}
SPL {X  -159.887, Y  +677.230, Z    +0.000, E1   -48.811, E3 +328474.504}
SPL {X  -159.602, Y  +682.629, Z    +0.000, E1   -48.761, E3 +328484.837}
SPL {X  -159.150, Y  +687.876, Z    +0.000, E1   -48.673, E3 +328495.076}
SPL {X  -158.569, Y  +692.776, Z    +0.000, E1   -48.570, E3 +328504.784}
SPL {X  -157.870, Y  +697.458, Z    +0.000, E1   -48.439, E3 +328514.213}
SPL {X  -157.028, Y  +702.144, Z    +0.000, E1   -48.297, E3 +328523.761}
SPL {X  -155.977, Y  +707.110, Z    +0.000, E1   -48.106, E3 +328534.065}
SPL {X  -154.657, Y  +712.464, Z    +0.000, E1   -47.874, E3 +328545.349}
SPL {X  -153.406, Y  +716.924, Z    +0.000, E1   -47.628, E3 +328554.915}
SPL {X  -152.020, Y  +721.367, Z    +0.000, E1   -47.374, E3 +328564.566}
SPL {X  -150.440, Y  +725.947, Z    +0.000, E1   -47.070, E3 +328574.671}
SPL {X  -148.730, Y  +730.459, Z    +0.000, E1   -46.749, E3 +328584.722}
SPL {X  -147.178, Y  +734.233, Z    +0.000, E1   -46.439, E3 +328593.256}
SPL {X  -140.222, Y  +748.536, Z    +0.000, E1   -42.074, E3 +328658.232}
ENDSPLINE

SPLINE
SPL {X  -152.021, Y  +721.365, Z    +0.000, E1   -28.339, E3 +328733.623}
SPL {X  -157.542, Y  +699.382, Z    +0.000, E1   -18.086, E3 +328749.141}
SPL {X  -159.386, Y  +685.393, Z    +0.000, E1   -10.664, E3 +328754.095}
SPL {X  -159.928, Y  +675.946, Z    +0.000, E1    -5.007, E3 +328756.134}
SPL {X  -159.990, Y  +671.468, Z    +0.000, E1    -2.030, E3 +328756.730}
SPL {X  -159.990, Y  +667.678, Z    +0.000, E1    +0.783, E3 +328757.080}
SPL {X  -159.990, Y  +663.139, Z    +0.000, E1    +5.135, E3 +328757.597}
SPL {X  -159.990, Y  +658.551, Z    +0.000, E1   +10.313, E3 +328758.371}
SPL {X  -159.990, Y  +653.526, Z    +0.000, E1   +16.156, E3 +328759.606}
SPL {X  -159.990, Y  +644.434, Z    +0.000, E1   +25.921, E3 +328762.801}
SPL {X  -159.990, Y  +612.255, Z    +0.000, E1   +44.102, E3 +328784.682}
SPL {X  -159.990, Y  +561.053, Z    +0.000, E1   +49.668, E3 +328849.515}
SPL {X  -159.990, Y  +552.984, Z    +0.000, E1   +49.619, E3 +328864.156}
SPL {X  -159.990, Y  +545.715, Z    +0.000, E1   +49.644, E3 +328877.240}
SPL {X  -159.990, Y  +537.339, Z    +0.000, E1   +49.638, E3 +328892.351}
SPL {X  -159.990, Y  +531.096, Z    +0.000, E1   +49.613, E3 +328903.649}
SPL {X  -159.990, Y  +524.316, Z    +0.000, E1   +49.648, E3 +328915.819}
SPL {X  -159.990, Y  +517.666, Z    +0.000, E1   +49.614, E3 +328927.880}
SPL {X  -159.990, Y  +511.038, Z    +0.000, E1   +49.636, E3 +328939.832}
SPL {X  -159.990, Y  +504.119, Z    +0.000, E1   +49.329, E3 +328954.215}
ENDSPLINE

SPLINE
SPL {X  -159.990, Y  +518.841, Z    +0.000, E1   +41.643, E3 +328969.543}
ENDSPLINE

SPLINE
SPL {X  -159.990, Y  +508.096, Z    +0.000, E1   +42.952, E3 +328986.810}
SPL {X  -159.990, Y  +500.642, Z    +0.000, E1   +43.747, E3 +328998.731}
SPL {X  -159.990, Y  +495.820, Z    +0.000, E1   +44.207, E3 +329006.618}
SPL {X  -159.990, Y  +487.435, Z    +0.000, E1   +45.185, E3 +329018.910}
SPL {X  -159.990, Y  +477.648, Z    +0.000, E1   +46.080, E3 +329033.907}
SPL {X  -159.990, Y  +469.952, Z    +0.000, E1   +46.750, E3 +329045.415}
SPL {X  -159.990, Y  +462.892, Z    +0.000, E1   +47.497, E3 +329054.899}
SPL {X  -159.990, Y  +452.841, Z    +0.000, E1   +48.572, E3 +329067.746}
SPL {X  -159.990, Y  +441.023, Z    +0.000, E1   +49.655, E3 +329082.997}
SPL {X  -159.990, Y  +431.096, Z    +0.000, E1   +50.075, E3 +329098.285}
SPL {X  -159.990, Y  +423.834, Z    +0.000, E1   +50.037, E3 +329111.258}
SPL {X  -159.990, Y  +417.693, Z    +0.000, E1   +50.049, E3 +329122.156}
SPL {X  -159.990, Y  +411.447, Z    +0.000, E1   +50.039, E3 +329133.275}
SPL {X  -159.990, Y  +403.654, Z    +0.000, E1   +50.076, E3 +329147.065}
SPL {X  -159.990, Y  +394.612, Z    +0.000, E1   +50.064, E3 +329163.153}
SPL {X  -159.990, Y  +387.356, Z    +0.000, E1   +50.042, E3 +329176.100}
SPL {X  -159.990, Y  +382.225, Z    +0.000, E1   +50.028, E3 +329185.245}
SPL {X  -159.846, Y  +375.718, Z    +0.000, E1   +50.041, E3 +329196.901}
SPL {X  -159.300, Y  +367.653, Z    +0.000, E1   +49.944, E3 +329211.809}
SPL {X  -158.412, Y  +360.086, Z    +0.000, E1   +49.787, E3 +329226.191}
SPL {X  -157.354, Y  +353.576, Z    +0.000, E1   +49.583, E3 +329238.894}
SPL {X  -156.029, Y  +347.121, Z    +0.000, E1   +49.358, E3 +329251.711}
SPL {X  -154.686, Y  +341.646, Z    +0.000, E1   +49.094, E3 +329262.855}
SPL {X  -153.439, Y  +337.188, Z    +0.000, E1   +48.857, E3 +329272.062}
SPL {X  -151.836, Y  +332.074, Z    +0.000, E1   +48.585, E3 +329282.738}
SPL {X  -150.221, Y  +327.451, Z    +0.000, E1   +48.251, E3 +329292.616}
SPL {X  -148.587, Y  +323.181, Z    +0.000, E1   +47.960, E3 +329301.800}
SPL {X  -146.510, Y  +318.222, Z    +0.000, E1   +47.558, E3 +329312.636}
SPL {X  -141.189, Y  +307.250, Z    +0.000, E1   +40.067, E3 +329398.810}
ENDSPLINE

SPLINE
SPL {X  -154.923, Y  +342.556, Z    +0.000, E1   +23.930, E3 +329460.309}
SPL {X  -158.138, Y  +358.230, Z    +0.000, E1   +16.243, E3 +329469.267}
SPL {X  -159.647, Y  +372.034, Z    +0.000, E1    +8.739, E3 +329473.631}
SPL {X  -159.989, Y  +381.927, Z    +0.000, E1    +2.565, E3 +329475.391}
SPL {X  -159.990, Y  +386.909, Z    +0.000, E1    -1.211, E3 +329475.934}
SPL {X  -159.990, Y  +390.921, Z    +0.000, E1    -5.111, E3 +329476.413}
SPL {X  -159.990, Y  +395.719, Z    +0.000, E1   -10.396, E3 +329477.232}
SPL {X  -159.990, Y  +400.739, Z    +0.000, E1   -16.236, E3 +329478.430}
SPL {X  -159.990, Y  +409.482, Z    +0.000, E1   -25.418, E3 +329481.635}
SPL {X  -159.990, Y  +440.741, Z    +0.000, E1   -43.570, E3 +329502.292}
SPL {X  -159.990, Y  +489.732, Z    +0.000, E1   -48.863, E3 +329566.450}
SPL {X  -159.990, Y  +496.901, Z    +0.000, E1   -48.832, E3 +329579.797}
SPL {X  -159.990, Y  +502.531, Z    +0.000, E1   -48.834, E3 +329590.242}
SPL {X  -159.990, Y  +508.013, Z    +0.000, E1   -48.835, E3 +329600.377}
SPL {X  -159.990, Y  +513.813, Z    +0.000, E1   -48.843, E3 +329611.125}
SPL {X  -159.990, Y  +522.177, Z    +0.000, E1   -48.881, E3 +329626.602}
SPL {X  -159.990, Y  +532.076, Z    +0.000, E1   -48.872, E3 +329644.975}
SPL {X  -159.990, Y  +539.248, Z    +0.000, E1   -48.832, E3 +329658.343}
SPL {X  -159.990, Y  +544.926, Z    +0.000, E1   -48.835, E3 +329668.872}
SPL {X  -159.990, Y  +550.252, Z    +0.000, E1   -48.827, E3 +329678.778}
SPL {X  -159.990, Y  +555.692, Z    +0.000, E1   -48.830, E3 +329688.875}
SPL {X  -159.990, Y  +561.308, Z    +0.000, E1   -48.827, E3 +329699.322}
SPL {X  -159.990, Y  +566.669, Z    +0.000, E1   -48.820, E3 +329709.271}
SPL {X  -159.990, Y  +572.248, Z    +0.000, E1   -48.830, E3 +329719.616}
SPL {X  -159.990, Y  +577.770, Z    +0.000, E1   -48.821, E3 +329729.863}
SPL {X  -159.990, Y  +583.108, Z    +0.000, E1   -48.828, E3 +329739.765}
SPL {X  -159.990, Y  +588.804, Z    +0.000, E1   -48.829, E3 +329750.322}
SPL {X  -159.990, Y  +594.280, Z    +0.000, E1   -48.826, E3 +329760.484}
SPL {X  -159.990, Y  +600.107, Z    +0.000, E1   -48.833, E3 +329771.298}
SPL {X  -159.990, Y  +605.910, Z    +0.000, E1   -48.823, E3 +329782.077}
SPL {X  -159.990, Y  +611.566, Z    +0.000, E1   -48.829, E3 +329792.566}
SPL {X  -159.990, Y  +617.357, Z    +0.000, E1   -48.824, E3 +329803.321}
SPL {X  -159.990, Y  +622.965, Z    +0.000, E1   -48.826, E3 +329813.720}
SPL {X  -159.990, Y  +629.255, Z    +0.000, E1   -48.834, E3 +329825.387}
SPL {X  -159.990, Y  +634.905, Z    +0.000, E1   -48.821, E3 +329835.884}
SPL {X  -159.990, Y  +640.372, Z    +0.000, E1   -48.828, E3 +329846.021}
SPL {X  -159.990, Y  +646.939, Z    +0.000, E1   -48.838, E3 +329858.191}
SPL {X  -159.990, Y  +653.448, Z    +0.000, E1   -48.827, E3 +329870.286}
SPL {X  -159.990, Y  +659.039, Z    +0.000, E1   -48.826, E3 +329880.650}
SPL {X  -159.990, Y  +664.817, Z    +0.000, E1   -48.832, E3 +329891.365}
SPL {X  -159.990, Y  +671.221, Z    +0.000, E1   -48.836, E3 +329903.238}
SPL {X  -159.887, Y  +677.230, Z    +0.000, E1   -48.811, E3 +329914.504}
SPL {X  -159.602, Y  +682.629, Z    +0.000, E1   -48.761, E3 +329924.837}
SPL {X  -159.150, Y  +687.876, Z    +0.000, E1   -48.673, E3 +329935.076}
SPL {X  -158.569, Y  +692.776, Z    +0.000, E1   -48.570, E3 +329944.784}
SPL {X  -157.870, Y  +697.458, Z    +0.000, E1   -48.439, E3 +329954.213}
SPL {X  -157.028, Y  +702.144, Z    +0.000, E1   -48.297, E3 +329963.761}
SPL {X  -155.977, Y  +707.110, Z    +0.000, E1   -48.106, E3 +329974.065}
SPL {X  -154.657, Y  +712.464, Z    +0.000, E1   -47.874, E3 +329985.349}
SPL {X  -153.406, Y  +716.924, Z    +0.000, E1   -47.628, E3 +329994.915}
SPL {X  -152.020, Y  +721.367, Z    +0.000, E1   -47.374, E3 +330004.566}
SPL {X  -150.440, Y  +725.947, Z    +0.000, E1   -47.070, E3 +330014.671}
SPL {X  -148.730, Y  +730.459, Z    +0.000, E1   -46.749, E3 +330024.722}
SPL {X  -147.178, Y  +734.233, Z    +0.000, E1   -46.439, E3 +330033.256}
SPL {X  -140.222, Y  +748.536, Z    +0.000, E1   -42.074, E3 +330098.232}
ENDSPLINE

SPLINE
SPL {X  -152.021, Y  +721.365, Z    +0.000, E1   -28.339, E3 +330173.623}
SPL {X  -158.165, Y  +695.595, Z    +0.000, E1   -16.189, E3 +330190.706}
SPL {X  -159.572, Y  +683.063, Z    +0.000, E1    -9.282, E3 +330194.713}
SPL {X  -159.928, Y  +675.946, Z    +0.000, E1    -5.007, E3 +330196.134}
SPL {X  -159.990, Y  +669.697, Z    +0.000, E1    -0.851, E3 +330196.894}
SPL {X  -159.990, Y  +665.698, Z    +0.000, E1    +2.616, E3 +330197.273}
SPL {X  -159.990, Y  +660.480, Z    +0.000, E1    +7.942, E3 +330198.031}
SPL {X  -159.990, Y  +653.526, Z    +0.000, E1   +16.156, E3 +330199.606}
SPL {X  -159.990, Y  +644.434, Z    +0.000, E1   +25.921, E3 +330202.801}
SPL {X  -159.990, Y  +612.255, Z    +0.000, E1   +44.102, E3 +330224.682}
SPL {X  -159.990, Y  +562.879, Z    +0.000, E1   +49.634, E3 +330286.271}
SPL {X  -159.990, Y  +554.544, Z    +0.000, E1   +49.649, E3 +330301.296}
SPL {X  -159.990, Y  +547.278, Z    +0.000, E1   +49.619, E3 +330314.455}
SPL {X  -159.990, Y  +540.489, Z    +0.000, E1   +49.634, E3 +330326.681}
SPL {X  -159.990, Y  +530.983, Z    +0.000, E1   +49.676, E3 +330343.752}
SPL {X  -159.990, Y  +522.804, Z    +0.000, E1   +49.620, E3 +330358.592}
SPL {X  -159.990, Y  +515.173, Z    +0.000, E1   +49.653, E3 +330372.330}
SPL {X  -159.990, Y  +505.472, Z    +0.000, E1   +49.465, E3 +330391.135}
ENDSPLINE

SPLINE
SPL {X  -159.990, Y  +518.841, Z    +0.000, E1   +41.643, E3 +330409.543}
ENDSPLINE

SPLINE
SPL {X  -159.990, Y  +508.096, Z    +0.000, E1   +42.952, E3 +330426.810}
SPL {X  -159.990, Y  +500.642, Z    +0.000, E1   +43.747, E3 +330438.731}
SPL {X  -159.990, Y  +495.820, Z    +0.000, E1   +44.207, E3 +330446.618}
SPL {X  -159.990, Y  +487.435, Z    +0.000, E1   +45.185, E3 +330458.910}
SPL {X  -159.990, Y  +477.648, Z    +0.000, E1   +46.080, E3 +330473.907}
SPL {X  -159.990, Y  +469.952, Z    +0.000, E1   +46.750, E3 +330485.415}
SPL {X  -159.990, Y  +460.762, Z    +0.000, E1   +47.755, E3 +330497.551}
SPL {X  -159.990, Y  +451.028, Z    +0.000, E1   +48.723, E3 +330510.163}
SPL {X  -159.990, Y  +441.023, Z    +0.000, E1   +49.655, E3 +330522.997}
SPL {X  -159.990, Y  +431.096, Z    +0.000, E1   +50.075, E3 +330538.285}
SPL {X  -159.990, Y  +423.834, Z    +0.000, E1   +50.037, E3 +330551.258}
SPL {X  -159.990, Y  +417.693, Z    +0.000, E1   +50.049, E3 +330562.156}
SPL {X  -159.990, Y  +411.447, Z    +0.000, E1   +50.039, E3 +330573.275}
SPL {X  -159.990, Y  +406.170, Z    +0.000, E1   +50.036, E3 +330582.647}
SPL {X  -159.990, Y  +399.787, Z    +0.000, E1   +50.064, E3 +330593.955}
SPL {X  -159.990, Y  +393.038, Z    +0.000, E1   +50.038, E3 +330605.989}
SPL {X  -159.990, Y  +387.356, Z    +0.000, E1   +50.042, E3 +330616.100}
SPL {X  -159.956, Y  +379.183, Z    +0.000, E1   +50.071, E3 +330630.614}
SPL {X  -159.413, Y  +368.921, Z    +0.000, E1   +49.998, E3 +330649.389}
SPL {X  -158.412, Y  +360.086, Z    +0.000, E1   +49.787, E3 +330666.191}
SPL {X  -157.077, Y  +352.107, Z    +0.000, E1   +49.567, E3 +330681.742}
SPL {X  -155.744, Y  +345.884, Z    +0.000, E1   +49.283, E3 +330694.229}
SPL {X  -154.686, Y  +341.646, Z    +0.000, E1   +49.094, E3 +330702.855}
SPL {X  -153.089, Y  +336.017, Z    +0.000, E1   +48.817, E3 +330714.464}
SPL {X  -151.481, Y  +331.019, Z    +0.000, E1   +48.491, E3 +330725.012}
SPL {X  -149.787, Y  +326.281, Z    +0.000, E1   +48.192, E3 +330735.100}
SPL {X  -148.124, Y  +322.035, Z    +0.000, E1   +47.846, E3 +330744.324}
SPL {X  -146.510, Y  +318.222, Z    +0.000, E1   +47.558, E3 +330752.636}
SPL {X  -141.189, Y  +307.250, Z    +0.000, E1   +40.067, E3 +330838.810}
ENDSPLINE

SPLINE
SPL {X  -154.923, Y  +342.556, Z    +0.000, E1   +23.930, E3 +330900.309}
SPL {X  -158.138, Y  +358.230, Z    +0.000, E1   +16.243, E3 +330909.267}
SPL {X  -159.407, Y  +368.849, Z    +0.000, E1   +10.504, E3 +330912.867}
SPL {X  -159.931, Y  +378.162, Z    +0.000, E1    +5.020, E3 +330914.852}
SPL {X  -159.990, Y  +384.616, Z    +0.000, E1    +0.627, E3 +330915.691}
SPL {X  -159.990, Y  +387.962, Z    +0.000, E1    -2.241, E3 +330916.048}
SPL {X  -159.990, Y  +390.921, Z    +0.000, E1    -5.111, E3 +330916.413}
SPL {X  -159.990, Y  +395.719, Z    +0.000, E1   -10.396, E3 +330917.232}
SPL {X  -159.990, Y  +400.739, Z    +0.000, E1   -16.236, E3 +330918.430}
SPL {X  -159.990, Y  +407.669, Z    +0.000, E1   -23.731, E3 +330920.753}
SPL {X  -159.990, Y  +417.102, Z    +0.000, E1   -32.094, E3 +330925.313}
SPL {X  -159.990, Y  +440.741, Z    +0.000, E1   -43.570, E3 +330942.292}
SPL {X  -159.990, Y  +488.072, Z    +0.000, E1   -48.834, E3 +331003.414}
SPL {X  -159.990, Y  +495.397, Z    +0.000, E1   -48.860, E3 +331016.963}
SPL {X  -159.990, Y  +502.531, Z    +0.000, E1   -48.834, E3 +331030.242}
SPL {X  -159.990, Y  +508.013, Z    +0.000, E1   -48.835, E3 +331040.377}
SPL {X  -159.990, Y  +513.813, Z    +0.000, E1   -48.843, E3 +331051.125}
SPL {X  -159.990, Y  +522.177, Z    +0.000, E1   -48.881, E3 +331066.602}
SPL {X  -159.990, Y  +532.076, Z    +0.000, E1   -48.872, E3 +331084.975}
SPL {X  -159.990, Y  +539.248, Z    +0.000, E1   -48.832, E3 +331098.343}
SPL {X  -159.990, Y  +544.926, Z    +0.000, E1   -48.835, E3 +331108.872}
SPL {X  -159.990, Y  +550.252, Z    +0.000, E1   -48.827, E3 +331118.778}
SPL {X  -159.990, Y  +555.692, Z    +0.000, E1   -48.830, E3 +331128.875}
SPL {X  -159.990, Y  +561.308, Z    +0.000, E1   -48.827, E3 +331139.322}
SPL {X  -159.990, Y  +566.669, Z    +0.000, E1   -48.820, E3 +331149.271}
SPL {X  -159.990, Y  +572.248, Z    +0.000, E1   -48.830, E3 +331159.616}
SPL {X  -159.990, Y  +577.770, Z    +0.000, E1   -48.821, E3 +331169.863}
SPL {X  -159.990, Y  +583.108, Z    +0.000, E1   -48.828, E3 +331179.765}
SPL {X  -159.990, Y  +588.804, Z    +0.000, E1   -48.829, E3 +331190.322}
SPL {X  -159.990, Y  +594.280, Z    +0.000, E1   -48.826, E3 +331200.484}
SPL {X  -159.990, Y  +600.107, Z    +0.000, E1   -48.833, E3 +331211.298}
SPL {X  -159.990, Y  +605.910, Z    +0.000, E1   -48.823, E3 +331222.077}
SPL {X  -159.990, Y  +611.566, Z    +0.000, E1   -48.829, E3 +331232.566}
SPL {X  -159.990, Y  +617.357, Z    +0.000, E1   -48.824, E3 +331243.321}
SPL {X  -159.990, Y  +622.965, Z    +0.000, E1   -48.826, E3 +331253.720}
SPL {X  -159.990, Y  +629.255, Z    +0.000, E1   -48.834, E3 +331265.387}
SPL {X  -159.990, Y  +634.905, Z    +0.000, E1   -48.821, E3 +331275.884}
SPL {X  -159.990, Y  +640.372, Z    +0.000, E1   -48.828, E3 +331286.021}
SPL {X  -159.990, Y  +646.939, Z    +0.000, E1   -48.838, E3 +331298.191}
SPL {X  -159.990, Y  +653.448, Z    +0.000, E1   -48.827, E3 +331310.286}
SPL {X  -159.990, Y  +659.039, Z    +0.000, E1   -48.826, E3 +331320.650}
SPL {X  -159.990, Y  +664.817, Z    +0.000, E1   -48.832, E3 +331331.365}
SPL {X  -159.990, Y  +671.221, Z    +0.000, E1   -48.836, E3 +331343.238}
SPL {X  -159.887, Y  +677.230, Z    +0.000, E1   -48.811, E3 +331354.504}
SPL {X  -159.602, Y  +682.629, Z    +0.000, E1   -48.761, E3 +331364.837}
SPL {X  -159.150, Y  +687.876, Z    +0.000, E1   -48.673, E3 +331375.076}
SPL {X  -158.569, Y  +692.776, Z    +0.000, E1   -48.570, E3 +331384.784}
SPL {X  -157.870, Y  +697.458, Z    +0.000, E1   -48.439, E3 +331394.213}
SPL {X  -157.028, Y  +702.144, Z    +0.000, E1   -48.297, E3 +331403.761}
SPL {X  -155.977, Y  +707.110, Z    +0.000, E1   -48.106, E3 +331414.065}
SPL {X  -154.657, Y  +712.464, Z    +0.000, E1   -47.874, E3 +331425.349}
SPL {X  -153.406, Y  +716.924, Z    +0.000, E1   -47.628, E3 +331434.915}
SPL {X  -152.020, Y  +721.367, Z    +0.000, E1   -47.374, E3 +331444.566}
SPL {X  -150.440, Y  +725.947, Z    +0.000, E1   -47.070, E3 +331454.671}
SPL {X  -148.730, Y  +730.459, Z    +0.000, E1   -46.749, E3 +331464.722}
SPL {X  -147.178, Y  +734.233, Z    +0.000, E1   -46.439, E3 +331473.256}
SPL {X  -140.263, Y  +748.461, Z    +0.000, E1   -42.675, E3 +331531.594}
ENDSPLINE

SPLINE
SPL {X  -141.835, Y  +745.525, Z    +0.000, E1   -39.068, E3 +331563.595}
SPL {X  -152.406, Y  +720.176, Z    +0.000, E1   -27.814, E3 +331614.808}
SPL {X  -158.165, Y  +695.595, Z    +0.000, E1   -16.189, E3 +331630.706}
SPL {X  -159.572, Y  +683.063, Z    +0.000, E1    -9.282, E3 +331634.713}
SPL {X  -159.928, Y  +675.946, Z    +0.000, E1    -5.007, E3 +331636.134}
SPL {X  -159.990, Y  +669.697, Z    +0.000, E1    -0.851, E3 +331636.894}
SPL {X  -159.990, Y  +665.698, Z    +0.000, E1    +2.616, E3 +331637.273}
SPL {X  -159.990, Y  +660.480, Z    +0.000, E1    +7.942, E3 +331638.031}
SPL {X  -159.990, Y  +653.526, Z    +0.000, E1   +16.156, E3 +331639.606}
SPL {X  -159.990, Y  +644.434, Z    +0.000, E1   +25.921, E3 +331642.801}
SPL {X  -159.990, Y  +612.255, Z    +0.000, E1   +44.102, E3 +331664.682}
SPL {X  -159.990, Y  +561.053, Z    +0.000, E1   +49.668, E3 +331729.515}
SPL {X  -159.990, Y  +552.984, Z    +0.000, E1   +49.619, E3 +331744.156}
SPL {X  -159.990, Y  +547.278, Z    +0.000, E1   +49.619, E3 +331754.455}
SPL {X  -159.990, Y  +538.738, Z    +0.000, E1   +49.672, E3 +331769.779}
SPL {X  -159.990, Y  +529.436, Z    +0.000, E1   +49.638, E3 +331786.603}
SPL {X  -159.990, Y  +522.804, Z    +0.000, E1   +49.620, E3 +331798.592}
SPL {X  -159.990, Y  +515.173, Z    +0.000, E1   +49.653, E3 +331812.330}
SPL {X  -159.990, Y  +505.896, Z    +0.000, E1   +49.645, E3 +331829.105}
ENDSPLINE

SPLINE
SPL {X  -159.990, Y  +511.561, Z    +0.000, E1   +45.946, E3 +331839.627}
SPL {X  -159.990, Y  +519.903, Z    +0.000, E1   +41.465, E3 +331847.946}
ENDSPLINE

SPLINE
SPL {X  -159.990, Y  +512.735, Z    +0.000, E1   +42.369, E3 +331859.523}
SPL {X  -159.990, Y  +505.924, Z    +0.000, E1   +43.199, E3 +331870.181}
SPL {X  -159.990, Y  +497.983, Z    +0.000, E1   +44.027, E3 +331883.054}
SPL {X  -159.990, Y  +487.435, Z    +0.000, E1   +45.185, E3 +331898.910}
SPL {X  -159.990, Y  +477.648, Z    +0.000, E1   +46.080, E3 +331913.907}
SPL {X  -159.990, Y  +469.952, Z    +0.000, E1   +46.750, E3 +331925.415}
SPL {X  -159.990, Y  +462.892, Z    +0.000, E1   +47.497, E3 +331934.899}
SPL {X  -159.990, Y  +452.841, Z    +0.000, E1   +48.572, E3 +331947.746}
SPL {X  -159.990, Y  +439.038, Z    +0.000, E1   +49.804, E3 +331965.798}
SPL {X  -159.990, Y  +429.517, Z    +0.000, E1   +50.043, E3 +331981.146}
SPL {X  -159.990, Y  +423.834, Z    +0.000, E1   +50.037, E3 +331991.258}
SPL {X  -159.990, Y  +417.693, Z    +0.000, E1   +50.049, E3 +332002.156}
SPL {X  -159.990, Y  +411.447, Z    +0.000, E1   +50.039, E3 +332013.275}
SPL {X  -159.990, Y  +406.170, Z    +0.000, E1   +50.036, E3 +332022.647}
SPL {X  -159.990, Y  +399.787, Z    +0.000, E1   +50.064, E3 +332033.955}
SPL {X  -159.990, Y  +393.038, Z    +0.000, E1   +50.038, E3 +332045.989}
SPL {X  -159.990, Y  +387.356, Z    +0.000, E1   +50.042, E3 +332056.100}
SPL {X  -159.956, Y  +379.183, Z    +0.000, E1   +50.071, E3 +332070.614}
SPL {X  -159.413, Y  +368.921, Z    +0.000, E1   +49.998, E3 +332089.389}
SPL {X  -158.412, Y  +360.086, Z    +0.000, E1   +49.787, E3 +332106.191}
SPL {X  -157.077, Y  +352.107, Z    +0.000, E1   +49.567, E3 +332121.742}
SPL {X  -155.744, Y  +345.884, Z    +0.000, E1   +49.283, E3 +332134.229}
SPL {X  -154.686, Y  +341.646, Z    +0.000, E1   +49.094, E3 +332142.855}
SPL {X  -153.089, Y  +336.017, Z    +0.000, E1   +48.817, E3 +332154.464}
SPL {X  -151.481, Y  +331.019, Z    +0.000, E1   +48.491, E3 +332165.012}
SPL {X  -149.787, Y  +326.281, Z    +0.000, E1   +48.192, E3 +332175.100}
SPL {X  -148.124, Y  +322.035, Z    +0.000, E1   +47.846, E3 +332184.324}
SPL {X  -146.510, Y  +318.222, Z    +0.000, E1   +47.558, E3 +332192.636}
SPL {X  -141.189, Y  +307.250, Z    +0.000, E1   +40.067, E3 +332278.810}
ENDSPLINE

SPLINE
SPL {X  -154.923, Y  +342.556, Z    +0.000, E1   +23.930, E3 +332340.309}
SPL {X  -158.138, Y  +358.230, Z    +0.000, E1   +16.243, E3 +332349.267}
SPL {X  -159.407, Y  +368.849, Z    +0.000, E1   +10.504, E3 +332352.867}
SPL {X  -159.931, Y  +378.162, Z    +0.000, E1    +5.020, E3 +332354.852}
SPL {X  -159.990, Y  +384.616, Z    +0.000, E1    +0.627, E3 +332355.691}
SPL {X  -159.990, Y  +387.962, Z    +0.000, E1    -2.241, E3 +332356.048}
SPL {X  -159.990, Y  +390.921, Z    +0.000, E1    -5.111, E3 +332356.413}
SPL {X  -159.990, Y  +395.719, Z    +0.000, E1   -10.396, E3 +332357.232}
SPL {X  -159.990, Y  +400.739, Z    +0.000, E1   -16.236, E3 +332358.430}
SPL {X  -159.990, Y  +407.669, Z    +0.000, E1   -23.731, E3 +332360.753}
SPL {X  -159.990, Y  +417.102, Z    +0.000, E1   -32.094, E3 +332365.313}
SPL {X  -159.990, Y  +440.741, Z    +0.000, E1   -43.570, E3 +332382.292}
SPL {X  -159.990, Y  +488.072, Z    +0.000, E1   -48.834, E3 +332443.414}
SPL {X  -159.990, Y  +495.397, Z    +0.000, E1   -48.860, E3 +332456.963}
SPL {X  -159.990, Y  +502.531, Z    +0.000, E1   -48.834, E3 +332470.242}
SPL {X  -159.990, Y  +508.013, Z    +0.000, E1   -48.835, E3 +332480.377}
SPL {X  -159.990, Y  +513.813, Z    +0.000, E1   -48.843, E3 +332491.125}
SPL {X  -159.990, Y  +522.177, Z    +0.000, E1   -48.881, E3 +332506.602}
SPL {X  -159.990, Y  +532.076, Z    +0.000, E1   -48.872, E3 +332524.975}
SPL {X  -159.990, Y  +539.248, Z    +0.000, E1   -48.832, E3 +332538.343}
SPL {X  -159.990, Y  +544.926, Z    +0.000, E1   -48.835, E3 +332548.872}
SPL {X  -159.990, Y  +550.252, Z    +0.000, E1   -48.827, E3 +332558.778}
SPL {X  -159.990, Y  +555.692, Z    +0.000, E1   -48.830, E3 +332568.875}
SPL {X  -159.990, Y  +561.308, Z    +0.000, E1   -48.827, E3 +332579.322}
SPL {X  -159.990, Y  +566.669, Z    +0.000, E1   -48.820, E3 +332589.271}
SPL {X  -159.990, Y  +572.248, Z    +0.000, E1   -48.830, E3 +332599.616}
SPL {X  -159.990, Y  +577.770, Z    +0.000, E1   -48.821, E3 +332609.863}
SPL {X  -159.990, Y  +583.108, Z    +0.000, E1   -48.828, E3 +332619.765}
SPL {X  -159.990, Y  +588.804, Z    +0.000, E1   -48.829, E3 +332630.322}
SPL {X  -159.990, Y  +594.280, Z    +0.000, E1   -48.826, E3 +332640.484}
SPL {X  -159.990, Y  +600.107, Z    +0.000, E1   -48.833, E3 +332651.298}
SPL {X  -159.990, Y  +605.910, Z    +0.000, E1   -48.823, E3 +332662.077}
SPL {X  -159.990, Y  +611.566, Z    +0.000, E1   -48.829, E3 +332672.566}
SPL {X  -159.990, Y  +617.357, Z    +0.000, E1   -48.824, E3 +332683.321}
SPL {X  -159.990, Y  +622.965, Z    +0.000, E1   -48.826, E3 +332693.720}
SPL {X  -159.990, Y  +629.255, Z    +0.000, E1   -48.834, E3 +332705.387}
SPL {X  -159.990, Y  +634.905, Z    +0.000, E1   -48.821, E3 +332715.884}
SPL {X  -159.990, Y  +640.372, Z    +0.000, E1   -48.828, E3 +332726.021}
SPL {X  -159.990, Y  +646.939, Z    +0.000, E1   -48.838, E3 +332738.191}
SPL {X  -159.990, Y  +653.448, Z    +0.000, E1   -48.827, E3 +332750.286}
SPL {X  -159.990, Y  +659.039, Z    +0.000, E1   -48.826, E3 +332760.650}
SPL {X  -159.990, Y  +664.817, Z    +0.000, E1   -48.832, E3 +332771.365}
SPL {X  -159.990, Y  +671.221, Z    +0.000, E1   -48.836, E3 +332783.238}
SPL {X  -159.887, Y  +677.230, Z    +0.000, E1   -48.811, E3 +332794.504}
SPL {X  -159.602, Y  +682.629, Z    +0.000, E1   -48.761, E3 +332804.837}
SPL {X  -159.150, Y  +687.876, Z    +0.000, E1   -48.673, E3 +332815.076}
SPL {X  -158.569, Y  +692.776, Z    +0.000, E1   -48.570, E3 +332824.784}
SPL {X  -157.870, Y  +697.458, Z    +0.000, E1   -48.439, E3 +332834.213}
SPL {X  -157.028, Y  +702.144, Z    +0.000, E1   -48.297, E3 +332843.761}
SPL {X  -155.977, Y  +707.110, Z    +0.000, E1   -48.106, E3 +332854.065}
SPL {X  -154.657, Y  +712.464, Z    +0.000, E1   -47.874, E3 +332865.349}
SPL {X  -153.406, Y  +716.924, Z    +0.000, E1   -47.628, E3 +332874.915}
SPL {X  -152.020, Y  +721.367, Z    +0.000, E1   -47.374, E3 +332884.566}
SPL {X  -150.440, Y  +725.947, Z    +0.000, E1   -47.070, E3 +332894.671}
SPL {X  -148.730, Y  +730.459, Z    +0.000, E1   -46.749, E3 +332904.722}
SPL {X  -147.178, Y  +734.233, Z    +0.000, E1   -46.439, E3 +332913.256}
SPL {X  -140.263, Y  +748.461, Z    +0.000, E1   -42.675, E3 +332971.594}
ENDSPLINE

SPLINE
SPL {X  -141.835, Y  +745.525, Z    +0.000, E1   -39.068, E3 +333003.595}
SPL {X  -152.406, Y  +720.176, Z    +0.000, E1   -27.814, E3 +333054.808}
SPL {X  -158.165, Y  +695.595, Z    +0.000, E1   -16.189, E3 +333070.706}
SPL {X  -159.572, Y  +683.063, Z    +0.000, E1    -9.282, E3 +333074.713}
SPL {X  -159.928, Y  +675.946, Z    +0.000, E1    -5.007, E3 +333076.134}
SPL {X  -159.990, Y  +669.697, Z    +0.000, E1    -0.851, E3 +333076.894}
SPL {X  -159.990, Y  +665.698, Z    +0.000, E1    +2.616, E3 +333077.273}
SPL {X  -159.990, Y  +660.480, Z    +0.000, E1    +7.942, E3 +333078.031}
SPL {X  -159.990, Y  +653.526, Z    +0.000, E1   +16.156, E3 +333079.606}
SPL {X  -159.990, Y  +644.434, Z    +0.000, E1   +25.921, E3 +333082.801}
SPL {X  -159.990, Y  +612.255, Z    +0.000, E1   +44.102, E3 +333104.682}
SPL {X  -159.990, Y  +561.053, Z    +0.000, E1   +49.668, E3 +333169.515}
SPL {X  -159.990, Y  +552.984, Z    +0.000, E1   +49.619, E3 +333184.156}
SPL {X  -159.990, Y  +547.278, Z    +0.000, E1   +49.619, E3 +333194.455}
SPL {X  -159.990, Y  +538.738, Z    +0.000, E1   +49.672, E3 +333209.779}
SPL {X  -159.990, Y  +529.436, Z    +0.000, E1   +49.638, E3 +333226.603}
SPL {X  -159.990, Y  +522.804, Z    +0.000, E1   +49.620, E3 +333238.592}
SPL {X  -159.990, Y  +515.173, Z    +0.000, E1   +49.653, E3 +333252.330}
SPL {X  -159.990, Y  +505.896, Z    +0.000, E1   +49.645, E3 +333269.105}
ENDSPLINE

SPLINE
SPL {X  -159.990, Y  +511.561, Z    +0.000, E1   +45.946, E3 +333279.627}
SPL {X  -159.990, Y  +519.903, Z    +0.000, E1   +41.465, E3 +333287.946}
ENDSPLINE

SPLINE
SPL {X  -159.990, Y  +512.735, Z    +0.000, E1   +42.369, E3 +333299.523}
SPL {X  -159.990, Y  +505.924, Z    +0.000, E1   +43.199, E3 +333310.181}
SPL {X  -159.990, Y  +497.983, Z    +0.000, E1   +44.027, E3 +333323.054}
SPL {X  -159.990, Y  +487.435, Z    +0.000, E1   +45.185, E3 +333338.910}
SPL {X  -159.990, Y  +477.648, Z    +0.000, E1   +46.080, E3 +333353.907}
SPL {X  -159.990, Y  +469.952, Z    +0.000, E1   +46.750, E3 +333365.415}
SPL {X  -159.990, Y  +462.892, Z    +0.000, E1   +47.497, E3 +333374.899}
SPL {X  -159.990, Y  +452.841, Z    +0.000, E1   +48.572, E3 +333387.746}
SPL {X  -159.990, Y  +439.038, Z    +0.000, E1   +49.804, E3 +333405.798}
SPL {X  -159.990, Y  +429.517, Z    +0.000, E1   +50.043, E3 +333421.146}
SPL {X  -159.990, Y  +423.834, Z    +0.000, E1   +50.037, E3 +333431.258}
SPL {X  -159.990, Y  +417.693, Z    +0.000, E1   +50.049, E3 +333442.156}
SPL {X  -159.990, Y  +411.447, Z    +0.000, E1   +50.039, E3 +333453.275}
SPL {X  -159.990, Y  +406.170, Z    +0.000, E1   +50.036, E3 +333462.647}
SPL {X  -159.990, Y  +399.787, Z    +0.000, E1   +50.064, E3 +333473.955}
SPL {X  -159.990, Y  +393.038, Z    +0.000, E1   +50.038, E3 +333485.989}
SPL {X  -159.990, Y  +387.356, Z    +0.000, E1   +50.042, E3 +333496.100}
SPL {X  -159.956, Y  +379.183, Z    +0.000, E1   +50.071, E3 +333510.614}
SPL {X  -159.413, Y  +368.921, Z    +0.000, E1   +49.998, E3 +333529.389}
SPL {X  -158.412, Y  +360.086, Z    +0.000, E1   +49.787, E3 +333546.191}
SPL {X  -157.077, Y  +352.107, Z    +0.000, E1   +49.567, E3 +333561.742}
SPL {X  -155.744, Y  +345.884, Z    +0.000, E1   +49.283, E3 +333574.229}
SPL {X  -154.686, Y  +341.646, Z    +0.000, E1   +49.094, E3 +333582.855}
SPL {X  -153.089, Y  +336.017, Z    +0.000, E1   +48.817, E3 +333594.464}
SPL {X  -151.481, Y  +331.019, Z    +0.000, E1   +48.491, E3 +333605.012}
SPL {X  -149.787, Y  +326.281, Z    +0.000, E1   +48.192, E3 +333615.100}
SPL {X  -148.124, Y  +322.035, Z    +0.000, E1   +47.846, E3 +333624.324}
SPL {X  -146.510, Y  +318.222, Z    +0.000, E1   +47.558, E3 +333632.636}
SPL {X  -141.189, Y  +307.250, Z    +0.000, E1   +40.067, E3 +333718.810}
ENDSPLINE

SPLINE
SPL {X  -154.923, Y  +342.556, Z    +0.000, E1   +23.930, E3 +333780.309}
SPL {X  -158.138, Y  +358.230, Z    +0.000, E1   +16.243, E3 +333789.267}
SPL {X  -159.407, Y  +368.849, Z    +0.000, E1   +10.504, E3 +333792.867}
SPL {X  -159.931, Y  +378.162, Z    +0.000, E1    +5.020, E3 +333794.852}
SPL {X  -159.990, Y  +384.616, Z    +0.000, E1    +0.627, E3 +333795.691}
SPL {X  -159.990, Y  +387.962, Z    +0.000, E1    -2.241, E3 +333796.048}
SPL {X  -159.990, Y  +390.921, Z    +0.000, E1    -5.111, E3 +333796.413}
SPL {X  -159.990, Y  +395.719, Z    +0.000, E1   -10.396, E3 +333797.232}
SPL {X  -159.990, Y  +400.739, Z    +0.000, E1   -16.236, E3 +333798.430}
SPL {X  -159.990, Y  +409.482, Z    +0.000, E1   -25.418, E3 +333801.635}
SPL {X  -159.990, Y  +440.741, Z    +0.000, E1   -43.570, E3 +333822.292}
SPL {X  -159.990, Y  +488.072, Z    +0.000, E1   -48.834, E3 +333883.414}
SPL {X  -159.990, Y  +495.397, Z    +0.000, E1   -48.860, E3 +333896.963}
SPL {X  -159.990, Y  +502.531, Z    +0.000, E1   -48.834, E3 +333910.242}
SPL {X  -159.990, Y  +508.013, Z    +0.000, E1   -48.835, E3 +333920.377}
SPL {X  -159.990, Y  +513.813, Z    +0.000, E1   -48.843, E3 +333931.125}
SPL {X  -159.990, Y  +522.177, Z    +0.000, E1   -48.881, E3 +333946.602}
SPL {X  -159.990, Y  +532.076, Z    +0.000, E1   -48.872, E3 +333964.975}
SPL {X  -159.990, Y  +539.248, Z    +0.000, E1   -48.832, E3 +333978.343}
SPL {X  -159.990, Y  +544.926, Z    +0.000, E1   -48.835, E3 +333988.872}
SPL {X  -159.990, Y  +550.252, Z    +0.000, E1   -48.827, E3 +333998.778}
SPL {X  -159.990, Y  +555.692, Z    +0.000, E1   -48.830, E3 +334008.875}
SPL {X  -159.990, Y  +561.308, Z    +0.000, E1   -48.827, E3 +334019.322}
SPL {X  -159.990, Y  +566.669, Z    +0.000, E1   -48.820, E3 +334029.271}
SPL {X  -159.990, Y  +572.248, Z    +0.000, E1   -48.830, E3 +334039.616}
SPL {X  -159.990, Y  +577.770, Z    +0.000, E1   -48.821, E3 +334049.863}
SPL {X  -159.990, Y  +583.108, Z    +0.000, E1   -48.828, E3 +334059.765}
SPL {X  -159.990, Y  +588.804, Z    +0.000, E1   -48.829, E3 +334070.322}
SPL {X  -159.990, Y  +594.280, Z    +0.000, E1   -48.826, E3 +334080.484}
SPL {X  -159.990, Y  +600.107, Z    +0.000, E1   -48.833, E3 +334091.298}
SPL {X  -159.990, Y  +605.910, Z    +0.000, E1   -48.823, E3 +334102.077}
SPL {X  -159.990, Y  +611.566, Z    +0.000, E1   -48.829, E3 +334112.566}
SPL {X  -159.990, Y  +617.357, Z    +0.000, E1   -48.824, E3 +334123.321}
SPL {X  -159.990, Y  +622.965, Z    +0.000, E1   -48.826, E3 +334133.720}
SPL {X  -159.990, Y  +629.255, Z    +0.000, E1   -48.834, E3 +334145.387}
SPL {X  -159.990, Y  +634.905, Z    +0.000, E1   -48.821, E3 +334155.884}
SPL {X  -159.990, Y  +640.372, Z    +0.000, E1   -48.828, E3 +334166.021}
SPL {X  -159.990, Y  +646.939, Z    +0.000, E1   -48.838, E3 +334178.191}
SPL {X  -159.990, Y  +653.448, Z    +0.000, E1   -48.827, E3 +334190.286}
SPL {X  -159.990, Y  +659.039, Z    +0.000, E1   -48.826, E3 +334200.650}
SPL {X  -159.990, Y  +664.817, Z    +0.000, E1   -48.832, E3 +334211.365}
SPL {X  -159.990, Y  +671.221, Z    +0.000, E1   -48.836, E3 +334223.238}
SPL {X  -159.887, Y  +677.230, Z    +0.000, E1   -48.811, E3 +334234.504}
SPL {X  -159.602, Y  +682.629, Z    +0.000, E1   -48.761, E3 +334244.837}
SPL {X  -159.150, Y  +687.876, Z    +0.000, E1   -48.673, E3 +334255.076}
SPL {X  -158.569, Y  +692.776, Z    +0.000, E1   -48.570, E3 +334264.784}
SPL {X  -157.870, Y  +697.458, Z    +0.000, E1   -48.439, E3 +334274.213}
SPL {X  -157.028, Y  +702.144, Z    +0.000, E1   -48.297, E3 +334283.761}
SPL {X  -155.977, Y  +707.110, Z    +0.000, E1   -48.106, E3 +334294.065}
SPL {X  -154.657, Y  +712.464, Z    +0.000, E1   -47.874, E3 +334305.349}
SPL {X  -153.406, Y  +716.924, Z    +0.000, E1   -47.628, E3 +334314.915}
SPL {X  -152.020, Y  +721.367, Z    +0.000, E1   -47.374, E3 +334324.566}
SPL {X  -150.440, Y  +725.947, Z    +0.000, E1   -47.070, E3 +334334.671}
SPL {X  -148.730, Y  +730.459, Z    +0.000, E1   -46.749, E3 +334344.722}
SPL {X  -147.178, Y  +734.233, Z    +0.000, E1   -46.439, E3 +334353.256}
SPL {X  -140.263, Y  +748.461, Z    +0.000, E1   -42.675, E3 +334411.594}
ENDSPLINE

SPLINE
SPL {X  -141.835, Y  +745.525, Z    +0.000, E1   -39.068, E3 +334443.595}
SPL {X  -152.406, Y  +720.176, Z    +0.000, E1   -27.814, E3 +334494.808}
SPL {X  -158.165, Y  +695.595, Z    +0.000, E1   -16.189, E3 +334510.706}
SPL {X  -159.572, Y  +683.063, Z    +0.000, E1    -9.282, E3 +334514.713}
SPL {X  -159.928, Y  +675.946, Z    +0.000, E1    -5.007, E3 +334516.134}
SPL {X  -159.990, Y  +671.468, Z    +0.000, E1    -2.030, E3 +334516.730}
SPL {X  -159.990, Y  +668.628, Z    +0.000, E1    +0.078, E3 +334516.994}
SPL {X  -159.990, Y  +665.698, Z    +0.000, E1    +2.616, E3 +334517.273}
SPL {X  -159.990, Y  +662.251, Z    +0.000, E1    +6.155, E3 +334517.719}
SPL {X  -159.990, Y  +658.551, Z    +0.000, E1   +10.313, E3 +334518.371}
SPL {X  -159.990, Y  +653.526, Z    +0.000, E1   +16.156, E3 +334519.606}
SPL {X  -159.990, Y  +644.434, Z    +0.000, E1   +25.921, E3 +334522.801}
SPL {X  -159.990, Y  +612.255, Z    +0.000, E1   +44.102, E3 +334544.682}
SPL {X  -159.990, Y  +561.053, Z    +0.000, E1   +49.668, E3 +334609.515}
SPL {X  -159.990, Y  +552.984, Z    +0.000, E1   +49.619, E3 +334624.156}
SPL {X  -159.990, Y  +545.715, Z    +0.000, E1   +49.644, E3 +334637.240}
SPL {X  -159.990, Y  +537.339, Z    +0.000, E1   +49.638, E3 +334652.351}
SPL {X  -159.990, Y  +531.096, Z    +0.000, E1   +49.613, E3 +334663.649}
SPL {X  -159.990, Y  +524.316, Z    +0.000, E1   +49.648, E3 +334675.819}
SPL {X  -159.990, Y  +515.173, Z    +0.000, E1   +49.653, E3 +334692.330}
SPL {X  -159.990, Y  +505.896, Z    +0.000, E1   +49.645, E3 +334709.105}
ENDSPLINE

SPLINE
SPL {X  -159.990, Y  +511.561, Z    +0.000, E1   +45.946, E3 +334719.627}
SPL {X  -159.990, Y  +519.903, Z    +0.000, E1   +41.465, E3 +334727.946}
ENDSPLINE

SPLINE
SPL {X  -159.990, Y  +512.735, Z    +0.000, E1   +42.369, E3 +334739.523}
SPL {X  -159.990, Y  +503.505, Z    +0.000, E1   +43.480, E3 +334754.068}
SPL {X  -159.990, Y  +495.820, Z    +0.000, E1   +44.207, E3 +334766.618}
SPL {X  -159.990, Y  +487.435, Z    +0.000, E1   +45.185, E3 +334778.910}
SPL {X  -159.990, Y  +477.648, Z    +0.000, E1   +46.080, E3 +334793.907}
SPL {X  -159.990, Y  +469.952, Z    +0.000, E1   +46.750, E3 +334805.415}
SPL {X  -159.990, Y  +460.762, Z    +0.000, E1   +47.755, E3 +334817.551}
SPL {X  -159.990, Y  +451.028, Z    +0.000, E1   +48.723, E3 +334830.163}
SPL {X  -159.990, Y  +441.023, Z    +0.000, E1   +49.655, E3 +334842.997}
SPL {X  -159.990, Y  +431.096, Z    +0.000, E1   +50.075, E3 +334858.285}
SPL {X  -159.990, Y  +423.834, Z    +0.000, E1   +50.037, E3 +334871.258}
SPL {X  -159.990, Y  +417.693, Z    +0.000, E1   +50.049, E3 +334882.156}
SPL {X  -159.990, Y  +408.922, Z    +0.000, E1   +50.085, E3 +334897.686}
SPL {X  -159.990, Y  +399.787, Z    +0.000, E1   +50.064, E3 +334913.955}
SPL {X  -159.990, Y  +393.038, Z    +0.000, E1   +50.038, E3 +334925.989}
SPL {X  -159.990, Y  +385.182, Z    +0.000, E1   +50.081, E3 +334939.906}
SPL {X  -159.846, Y  +375.718, Z    +0.000, E1   +50.041, E3 +334956.901}
SPL {X  -159.300, Y  +367.653, Z    +0.000, E1   +49.944, E3 +334971.809}
SPL {X  -158.412, Y  +360.086, Z    +0.000, E1   +49.787, E3 +334986.191}
SPL {X  -157.077, Y  +352.107, Z    +0.000, E1   +49.567, E3 +335001.742}
SPL {X  -155.744, Y  +345.884, Z    +0.000, E1   +49.283, E3 +335014.229}
SPL {X  -154.686, Y  +341.646, Z    +0.000, E1   +49.094, E3 +335022.855}
SPL {X  -153.089, Y  +336.017, Z    +0.000, E1   +48.817, E3 +335034.464}
SPL {X  -150.861, Y  +329.230, Z    +0.000, E1   +48.419, E3 +335048.753}
SPL {X  -148.587, Y  +323.181, Z    +0.000, E1   +47.960, E3 +335061.800}
SPL {X  -146.510, Y  +318.222, Z    +0.000, E1   +47.558, E3 +335072.636}
SPL {X  -141.189, Y  +307.250, Z    +0.000, E1   +40.067, E3 +335158.810}
ENDSPLINE

SPLINE
SPL {X  -154.923, Y  +342.556, Z    +0.000, E1   +23.930, E3 +335220.309}
SPL {X  -158.138, Y  +358.230, Z    +0.000, E1   +16.243, E3 +335229.267}
SPL {X  -159.407, Y  +368.849, Z    +0.000, E1   +10.504, E3 +335232.867}
SPL {X  -159.931, Y  +378.162, Z    +0.000, E1    +5.020, E3 +335234.852}
SPL {X  -159.990, Y  +384.616, Z    +0.000, E1    +0.627, E3 +335235.691}
SPL {X  -159.990, Y  +387.962, Z    +0.000, E1    -2.241, E3 +335236.048}
SPL {X  -159.990, Y  +390.921, Z    +0.000, E1    -5.111, E3 +335236.413}
SPL {X  -159.990, Y  +395.719, Z    +0.000, E1   -10.396, E3 +335237.232}
SPL {X  -159.990, Y  +400.739, Z    +0.000, E1   -16.236, E3 +335238.430}
SPL {X  -159.990, Y  +409.482, Z    +0.000, E1   -25.418, E3 +335241.635}
SPL {X  -159.990, Y  +440.741, Z    +0.000, E1   -43.570, E3 +335262.292}
SPL {X  -159.990, Y  +488.072, Z    +0.000, E1   -48.834, E3 +335323.414}
SPL {X  -159.990, Y  +495.397, Z    +0.000, E1   -48.860, E3 +335336.963}
SPL {X  -159.990, Y  +502.531, Z    +0.000, E1   -48.834, E3 +335350.242}
SPL {X  -159.990, Y  +508.013, Z    +0.000, E1   -48.835, E3 +335360.377}
SPL {X  -159.990, Y  +513.813, Z    +0.000, E1   -48.843, E3 +335371.125}
SPL {X  -159.990, Y  +522.177, Z    +0.000, E1   -48.881, E3 +335386.602}
SPL {X  -159.990, Y  +532.076, Z    +0.000, E1   -48.872, E3 +335404.975}
SPL {X  -159.990, Y  +539.248, Z    +0.000, E1   -48.832, E3 +335418.343}
SPL {X  -159.990, Y  +544.926, Z    +0.000, E1   -48.835, E3 +335428.872}
SPL {X  -159.990, Y  +550.252, Z    +0.000, E1   -48.827, E3 +335438.778}
SPL {X  -159.990, Y  +555.692, Z    +0.000, E1   -48.830, E3 +335448.875}
SPL {X  -159.990, Y  +561.308, Z    +0.000, E1   -48.827, E3 +335459.322}
SPL {X  -159.990, Y  +566.669, Z    +0.000, E1   -48.820, E3 +335469.271}
SPL {X  -159.990, Y  +572.248, Z    +0.000, E1   -48.830, E3 +335479.616}
SPL {X  -159.990, Y  +577.770, Z    +0.000, E1   -48.821, E3 +335489.863}
SPL {X  -159.990, Y  +583.108, Z    +0.000, E1   -48.828, E3 +335499.765}
SPL {X  -159.990, Y  +588.804, Z    +0.000, E1   -48.829, E3 +335510.322}
SPL {X  -159.990, Y  +594.280, Z    +0.000, E1   -48.826, E3 +335520.484}
SPL {X  -159.990, Y  +600.107, Z    +0.000, E1   -48.833, E3 +335531.298}
SPL {X  -159.990, Y  +605.910, Z    +0.000, E1   -48.823, E3 +335542.077}
SPL {X  -159.990, Y  +611.566, Z    +0.000, E1   -48.829, E3 +335552.566}
SPL {X  -159.990, Y  +617.357, Z    +0.000, E1   -48.824, E3 +335563.321}
SPL {X  -159.990, Y  +622.965, Z    +0.000, E1   -48.826, E3 +335573.720}
SPL {X  -159.990, Y  +629.255, Z    +0.000, E1   -48.834, E3 +335585.387}
SPL {X  -159.990, Y  +634.905, Z    +0.000, E1   -48.821, E3 +335595.884}
SPL {X  -159.990, Y  +640.372, Z    +0.000, E1   -48.828, E3 +335606.021}
SPL {X  -159.990, Y  +646.939, Z    +0.000, E1   -48.838, E3 +335618.191}
SPL {X  -159.990, Y  +653.448, Z    +0.000, E1   -48.827, E3 +335630.286}
SPL {X  -159.990, Y  +659.039, Z    +0.000, E1   -48.826, E3 +335640.650}
SPL {X  -159.990, Y  +664.817, Z    +0.000, E1   -48.832, E3 +335651.365}
SPL {X  -159.990, Y  +671.221, Z    +0.000, E1   -48.836, E3 +335663.238}
SPL {X  -159.887, Y  +677.230, Z    +0.000, E1   -48.811, E3 +335674.504}
SPL {X  -159.602, Y  +682.629, Z    +0.000, E1   -48.761, E3 +335684.837}
SPL {X  -159.150, Y  +687.876, Z    +0.000, E1   -48.673, E3 +335695.076}
SPL {X  -158.569, Y  +692.776, Z    +0.000, E1   -48.570, E3 +335704.784}
SPL {X  -157.870, Y  +697.458, Z    +0.000, E1   -48.439, E3 +335714.213}
SPL {X  -157.028, Y  +702.144, Z    +0.000, E1   -48.297, E3 +335723.761}
SPL {X  -155.977, Y  +707.110, Z    +0.000, E1   -48.106, E3 +335734.065}
SPL {X  -154.657, Y  +712.464, Z    +0.000, E1   -47.874, E3 +335745.349}
SPL {X  -153.406, Y  +716.924, Z    +0.000, E1   -47.628, E3 +335754.915}
SPL {X  -152.020, Y  +721.367, Z    +0.000, E1   -47.374, E3 +335764.566}
SPL {X  -150.440, Y  +725.947, Z    +0.000, E1   -47.070, E3 +335774.671}
SPL {X  -148.730, Y  +730.459, Z    +0.000, E1   -46.749, E3 +335784.722}
SPL {X  -147.178, Y  +734.233, Z    +0.000, E1   -46.439, E3 +335793.256}
SPL {X  -140.222, Y  +748.536, Z    +0.000, E1   -42.074, E3 +335858.232}
ENDSPLINE

SPLINE
SPL {X  -152.021, Y  +721.365, Z    +0.000, E1   -28.339, E3 +335933.623}
SPL {X  -158.165, Y  +695.595, Z    +0.000, E1   -16.189, E3 +335950.706}
SPL {X  -159.572, Y  +683.063, Z    +0.000, E1    -9.282, E3 +335954.713}
SPL {X  -159.928, Y  +675.946, Z    +0.000, E1    -5.007, E3 +335956.134}
SPL {X  -159.990, Y  +669.697, Z    +0.000, E1    -0.851, E3 +335956.894}
SPL {X  -159.990, Y  +665.698, Z    +0.000, E1    +2.616, E3 +335957.273}
SPL {X  -159.990, Y  +662.251, Z    +0.000, E1    +6.155, E3 +335957.719}
SPL {X  -159.990, Y  +658.551, Z    +0.000, E1   +10.313, E3 +335958.371}
SPL {X  -159.990, Y  +653.526, Z    +0.000, E1   +16.156, E3 +335959.606}
SPL {X  -159.990, Y  +644.434, Z    +0.000, E1   +25.921, E3 +335962.801}
SPL {X  -159.990, Y  +612.255, Z    +0.000, E1   +44.102, E3 +335984.682}
SPL {X  -159.990, Y  +561.053, Z    +0.000, E1   +49.668, E3 +336049.515}
SPL {X  -159.990, Y  +552.984, Z    +0.000, E1   +49.619, E3 +336064.156}
SPL {X  -159.990, Y  +547.278, Z    +0.000, E1   +49.619, E3 +336074.455}
SPL {X  -159.990, Y  +538.738, Z    +0.000, E1   +49.672, E3 +336089.779}
SPL {X  -159.990, Y  +529.436, Z    +0.000, E1   +49.638, E3 +336106.603}
SPL {X  -159.990, Y  +522.804, Z    +0.000, E1   +49.620, E3 +336118.592}
SPL {X  -159.990, Y  +515.173, Z    +0.000, E1   +49.653, E3 +336132.330}
SPL {X  -159.990, Y  +505.472, Z    +0.000, E1   +49.465, E3 +336151.135}
ENDSPLINE

SPLINE
SPL {X  -159.990, Y  +518.841, Z    +0.000, E1   +41.643, E3 +336169.543}
ENDSPLINE

SPLINE
SPL {X  -159.990, Y  +508.096, Z    +0.000, E1   +42.952, E3 +336186.810}
SPL {X  -159.990, Y  +500.642, Z    +0.000, E1   +43.747, E3 +336198.731}
SPL {X  -159.990, Y  +495.820, Z    +0.000, E1   +44.207, E3 +336206.618}
SPL {X  -159.990, Y  +487.435, Z    +0.000, E1   +45.185, E3 +336218.910}
SPL {X  -159.990, Y  +477.648, Z    +0.000, E1   +46.080, E3 +336233.907}
SPL {X  -159.990, Y  +469.952, Z    +0.000, E1   +46.750, E3 +336245.415}
SPL {X  -159.990, Y  +462.892, Z    +0.000, E1   +47.497, E3 +336254.899}
SPL {X  -159.990, Y  +452.841, Z    +0.000, E1   +48.572, E3 +336267.746}
SPL {X  -159.990, Y  +439.038, Z    +0.000, E1   +49.804, E3 +336285.798}
SPL {X  -159.990, Y  +429.517, Z    +0.000, E1   +50.043, E3 +336301.146}
SPL {X  -159.990, Y  +423.834, Z    +0.000, E1   +50.037, E3 +336311.258}
SPL {X  -159.990, Y  +417.693, Z    +0.000, E1   +50.049, E3 +336322.156}
SPL {X  -159.990, Y  +411.447, Z    +0.000, E1   +50.039, E3 +336333.275}
SPL {X  -159.990, Y  +406.170, Z    +0.000, E1   +50.036, E3 +336342.647}
SPL {X  -159.990, Y  +399.787, Z    +0.000, E1   +50.064, E3 +336353.955}
SPL {X  -159.990, Y  +393.038, Z    +0.000, E1   +50.038, E3 +336365.989}
SPL {X  -159.990, Y  +387.356, Z    +0.000, E1   +50.042, E3 +336376.100}
SPL {X  -159.990, Y  +382.225, Z    +0.000, E1   +50.028, E3 +336385.245}
SPL {X  -159.846, Y  +375.718, Z    +0.000, E1   +50.041, E3 +336396.901}
SPL {X  -159.443, Y  +369.277, Z    +0.000, E1   +49.941, E3 +336408.815}
SPL {X  -158.871, Y  +363.614, Z    +0.000, E1   +49.855, E3 +336419.459}
SPL {X  -158.179, Y  +358.495, Z    +0.000, E1   +49.715, E3 +336429.308}
SPL {X  -157.077, Y  +352.107, Z    +0.000, E1   +49.567, E3 +336441.742}
SPL {X  -155.744, Y  +345.884, Z    +0.000, E1   +49.283, E3 +336454.229}
SPL {X  -154.686, Y  +341.646, Z    +0.000, E1   +49.094, E3 +336462.855}
SPL {X  -153.439, Y  +337.188, Z    +0.000, E1   +48.857, E3 +336472.062}
SPL {X  -151.836, Y  +332.074, Z    +0.000, E1   +48.585, E3 +336482.738}
SPL {X  -150.221, Y  +327.451, Z    +0.000, E1   +48.251, E3 +336492.616}
SPL {X  -148.587, Y  +323.181, Z    +0.000, E1   +47.960, E3 +336501.800}
SPL {X  -146.510, Y  +318.222, Z    +0.000, E1   +47.558, E3 +336512.636}
SPL {X  -141.189, Y  +307.250, Z    +0.000, E1   +40.067, E3 +336598.810}
ENDSPLINE

SPLINE
SPL {X  -154.923, Y  +342.556, Z    +0.000, E1   +23.930, E3 +336660.309}
SPL {X  -158.138, Y  +358.230, Z    +0.000, E1   +16.243, E3 +336669.267}
SPL {X  -159.647, Y  +372.034, Z    +0.000, E1    +8.739, E3 +336673.631}
SPL {X  -159.989, Y  +381.927, Z    +0.000, E1    +2.565, E3 +336675.391}
SPL {X  -159.990, Y  +386.909, Z    +0.000, E1    -1.211, E3 +336675.934}
SPL {X  -159.990, Y  +390.921, Z    +0.000, E1    -5.111, E3 +336676.413}
SPL {X  -159.990, Y  +395.719, Z    +0.000, E1   -10.396, E3 +336677.232}
SPL {X  -159.990, Y  +400.739, Z    +0.000, E1   -16.236, E3 +336678.430}
SPL {X  -159.990, Y  +409.482, Z    +0.000, E1   -25.418, E3 +336681.635}
SPL {X  -159.990, Y  +440.741, Z    +0.000, E1   -43.570, E3 +336702.292}
SPL {X  -159.990, Y  +489.732, Z    +0.000, E1   -48.863, E3 +336766.450}
SPL {X  -159.990, Y  +496.901, Z    +0.000, E1   -48.832, E3 +336779.797}
SPL {X  -159.990, Y  +502.531, Z    +0.000, E1   -48.834, E3 +336790.242}
SPL {X  -159.990, Y  +508.013, Z    +0.000, E1   -48.835, E3 +336800.377}
SPL {X  -159.990, Y  +513.813, Z    +0.000, E1   -48.843, E3 +336811.125}
SPL {X  -159.990, Y  +522.177, Z    +0.000, E1   -48.881, E3 +336826.602}
SPL {X  -159.990, Y  +532.076, Z    +0.000, E1   -48.872, E3 +336844.975}
SPL {X  -159.990, Y  +539.248, Z    +0.000, E1   -48.832, E3 +336858.343}
SPL {X  -159.990, Y  +544.926, Z    +0.000, E1   -48.835, E3 +336868.872}
SPL {X  -159.990, Y  +550.252, Z    +0.000, E1   -48.827, E3 +336878.778}
SPL {X  -159.990, Y  +555.692, Z    +0.000, E1   -48.830, E3 +336888.875}
SPL {X  -159.990, Y  +561.308, Z    +0.000, E1   -48.827, E3 +336899.322}
SPL {X  -159.990, Y  +566.669, Z    +0.000, E1   -48.820, E3 +336909.271}
SPL {X  -159.990, Y  +572.248, Z    +0.000, E1   -48.830, E3 +336919.616}
SPL {X  -159.990, Y  +577.770, Z    +0.000, E1   -48.821, E3 +336929.863}
SPL {X  -159.990, Y  +583.108, Z    +0.000, E1   -48.828, E3 +336939.765}
SPL {X  -159.990, Y  +588.804, Z    +0.000, E1   -48.829, E3 +336950.322}
SPL {X  -159.990, Y  +594.280, Z    +0.000, E1   -48.826, E3 +336960.484}
SPL {X  -159.990, Y  +600.107, Z    +0.000, E1   -48.833, E3 +336971.298}
SPL {X  -159.990, Y  +605.910, Z    +0.000, E1   -48.823, E3 +336982.077}
SPL {X  -159.990, Y  +611.566, Z    +0.000, E1   -48.829, E3 +336992.566}
SPL {X  -159.990, Y  +617.357, Z    +0.000, E1   -48.824, E3 +337003.321}
SPL {X  -159.990, Y  +622.965, Z    +0.000, E1   -48.826, E3 +337013.720}
SPL {X  -159.990, Y  +629.255, Z    +0.000, E1   -48.834, E3 +337025.387}
SPL {X  -159.990, Y  +634.905, Z    +0.000, E1   -48.821, E3 +337035.884}
SPL {X  -159.990, Y  +640.372, Z    +0.000, E1   -48.828, E3 +337046.021}
SPL {X  -159.990, Y  +646.939, Z    +0.000, E1   -48.838, E3 +337058.191}
SPL {X  -159.990, Y  +653.448, Z    +0.000, E1   -48.827, E3 +337070.286}
SPL {X  -159.990, Y  +659.039, Z    +0.000, E1   -48.826, E3 +337080.650}
SPL {X  -159.990, Y  +664.817, Z    +0.000, E1   -48.832, E3 +337091.365}
SPL {X  -159.990, Y  +671.221, Z    +0.000, E1   -48.836, E3 +337103.238}
SPL {X  -159.887, Y  +677.230, Z    +0.000, E1   -48.811, E3 +337114.504}
SPL {X  -159.602, Y  +682.629, Z    +0.000, E1   -48.761, E3 +337124.837}
SPL {X  -159.150, Y  +687.876, Z    +0.000, E1   -48.673, E3 +337135.076}
SPL {X  -158.569, Y  +692.776, Z    +0.000, E1   -48.570, E3 +337144.784}
SPL {X  -157.870, Y  +697.458, Z    +0.000, E1   -48.439, E3 +337154.213}
SPL {X  -157.028, Y  +702.144, Z    +0.000, E1   -48.297, E3 +337163.761}
SPL {X  -155.977, Y  +707.110, Z    +0.000, E1   -48.106, E3 +337174.065}
SPL {X  -154.657, Y  +712.464, Z    +0.000, E1   -47.874, E3 +337185.349}
SPL {X  -153.406, Y  +716.924, Z    +0.000, E1   -47.628, E3 +337194.915}
SPL {X  -152.020, Y  +721.367, Z    +0.000, E1   -47.374, E3 +337204.566}
SPL {X  -150.440, Y  +725.947, Z    +0.000, E1   -47.070, E3 +337214.671}
SPL {X  -148.730, Y  +730.459, Z    +0.000, E1   -46.749, E3 +337224.722}
SPL {X  -147.178, Y  +734.233, Z    +0.000, E1   -46.439, E3 +337233.256}
SPL {X  -140.222, Y  +748.536, Z    +0.000, E1   -42.074, E3 +337298.232}
ENDSPLINE

SPLINE
SPL {X  -152.021, Y  +721.365, Z    +0.000, E1   -28.339, E3 +337373.623}
SPL {X  -157.542, Y  +699.382, Z    +0.000, E1   -18.086, E3 +337389.141}
SPL {X  -159.386, Y  +685.393, Z    +0.000, E1   -10.664, E3 +337394.095}
SPL {X  -159.928, Y  +675.946, Z    +0.000, E1    -5.007, E3 +337396.134}
SPL {X  -159.990, Y  +671.468, Z    +0.000, E1    -2.030, E3 +337396.730}
SPL {X  -159.990, Y  +668.628, Z    +0.000, E1    +0.078, E3 +337396.994}
SPL {X  -159.990, Y  +665.698, Z    +0.000, E1    +2.616, E3 +337397.273}
SPL {X  -159.990, Y  +662.251, Z    +0.000, E1    +6.155, E3 +337397.719}
SPL {X  -159.990, Y  +658.551, Z    +0.000, E1   +10.313, E3 +337398.371}
SPL {X  -159.990, Y  +653.526, Z    +0.000, E1   +16.156, E3 +337399.606}
SPL {X  -159.990, Y  +644.434, Z    +0.000, E1   +25.921, E3 +337402.801}
SPL {X  -159.990, Y  +612.255, Z    +0.000, E1   +44.102, E3 +337424.682}
SPL {X  -159.990, Y  +567.037, Z    +0.000, E1   +49.607, E3 +337478.826}
SPL {X  -159.990, Y  +562.169, Z    +0.000, E1   +49.620, E3 +337487.582}
SPL {X  -159.990, Y  +554.544, Z    +0.000, E1   +49.649, E3 +337501.296}
SPL {X  -159.990, Y  +545.715, Z    +0.000, E1   +49.644, E3 +337517.240}
SPL {X  -159.990, Y  +537.339, Z    +0.000, E1   +49.638, E3 +337532.351}
SPL {X  -159.990, Y  +529.436, Z    +0.000, E1   +49.638, E3 +337546.603}
SPL {X  -159.990, Y  +520.280, Z    +0.000, E1   +49.665, E3 +337563.082}
SPL {X  -159.990, Y  +511.038, Z    +0.000, E1   +49.636, E3 +337579.832}
SPL {X  -159.990, Y  +504.260, Z    +0.000, E1   +49.614, E3 +337592.105}
ENDSPLINE

SPLINE
SPL {X  -159.990, Y  +511.561, Z    +0.000, E1   +45.946, E3 +337599.627}
SPL {X  -159.990, Y  +518.175, Z    +0.000, E1   +41.708, E3 +337610.702}
ENDSPLINE

SPLINE
SPL {X  -159.990, Y  +508.096, Z    +0.000, E1   +42.952, E3 +337626.810}
SPL {X  -159.990, Y  +497.983, Z    +0.000, E1   +44.027, E3 +337643.054}
SPL {X  -159.990, Y  +487.435, Z    +0.000, E1   +45.185, E3 +337658.910}
SPL {X  -159.990, Y  +477.648, Z    +0.000, E1   +46.080, E3 +337673.907}
SPL {X  -159.990, Y  +469.952, Z    +0.000, E1   +46.750, E3 +337685.415}
SPL {X  -159.990, Y  +462.892, Z    +0.000, E1   +47.497, E3 +337694.899}
SPL {X  -159.990, Y  +452.841, Z    +0.000, E1   +48.572, E3 +337707.746}
SPL {X  -159.990, Y  +440.939, Z    +0.000, E1   +49.652, E3 +337723.177}
ENDSPLINE

SPLINE
SPL {X  -159.990, Y  +453.647, Z    +0.000, E1   +43.235, E3 +337735.339}
ENDSPLINE

SPLINE
SPL {X  -159.990, Y  +448.702, Z    +0.000, E1   +43.218, E3 +337746.568}
SPL {X  -159.990, Y  +444.476, Z    +0.000, E1   +43.219, E3 +337756.106}
SPL {X  -159.990, Y  +440.246, Z    +0.000, E1   +43.217, E3 +337765.664}
SPL {X  -159.990, Y  +434.411, Z    +0.000, E1   +43.246, E3 +337778.794}
SPL {X  -159.990, Y  +429.216, Z    +0.000, E1   +43.210, E3 +337790.567}
SPL {X  -159.990, Y  +424.433, Z    +0.000, E1   +43.237, E3 +337801.314}
SPL {X  -159.990, Y  +419.466, Z    +0.000, E1   +43.217, E3 +337812.554}
SPL {X  -159.990, Y  +414.585, Z    +0.000, E1   +43.233, E3 +337823.546}
SPL {X  -159.990, Y  +409.927, Z    +0.000, E1   +43.217, E3 +337834.078}
SPL {X  -159.990, Y  +405.428, Z    +0.000, E1   +43.230, E3 +337844.236}
SPL {X  -159.990, Y  +398.518, Z    +0.000, E1   +43.261, E3 +337859.790}
SPL {X  -159.990, Y  +392.163, Z    +0.000, E1   +43.223, E3 +337874.190}
SPL {X  -159.990, Y  +387.342, Z    +0.000, E1   +43.224, E3 +337885.068}
SPL {X  -159.990, Y  +382.548, Z    +0.000, E1   +43.224, E3 +337895.890}
SPL {X  -159.922, Y  +377.835, Z    +0.000, E1   +43.211, E3 +337906.607}
SPL {X  -159.712, Y  +373.072, Z    +0.000, E1   +43.177, E3 +337917.573}
SPL {X  -159.289, Y  +367.537, Z    +0.000, E1   +43.118, E3 +337930.485}
SPL {X  -158.730, Y  +362.464, Z    +0.000, E1   +43.003, E3 +337942.517}
SPL {X  -158.182, Y  +358.518, Z    +0.000, E1   +42.902, E3 +337951.995}
SPL {X  -157.507, Y  +354.423, Z    +0.000, E1   +42.786, E3 +337961.941}
SPL {X  -156.676, Y  +350.104, Z    +0.000, E1   +42.637, E3 +337972.546}
SPL {X  -155.807, Y  +346.154, Z    +0.000, E1   +42.470, E3 +337982.373}
SPL {X  -154.777, Y  +341.993, Z    +0.000, E1   +42.302, E3 +337992.798}
SPL {X  -153.585, Y  +337.686, Z    +0.000, E1   +42.062, E3 +338003.774}
SPL {X  -152.412, Y  +333.846, Z    +0.000, E1   +41.856, E3 +338013.616}
SPL {X  -151.009, Y  +329.651, Z    +0.000, E1   +41.581, E3 +338024.516}
SPL {X  -148.356, Y  +322.607, Z    +0.000, E1   +36.121, E3 +338084.992}
ENDSPLINE

SPLINE
SPL {X  -156.487, Y  +349.204, Z    +0.000, E1   +21.338, E3 +338140.117}
SPL {X  -159.136, Y  +365.992, Z    +0.000, E1   +12.463, E3 +338150.876}
SPL {X  -159.799, Y  +374.694, Z    +0.000, E1    +7.504, E3 +338153.980}
SPL {X  -159.976, Y  +380.404, Z    +0.000, E1    +3.959, E3 +338155.513}
SPL {X  -159.990, Y  +384.773, Z    +0.000, E1    +1.003, E3 +338156.407}
SPL {X  -159.990, Y  +387.968, Z    +0.000, E1    -1.448, E3 +338156.975}
SPL {X  -159.990, Y  +391.397, Z    +0.000, E1    -4.422, E3 +338157.599}
SPL {X  -159.990, Y  +395.864, Z    +0.000, E1    -8.712, E3 +338158.688}
SPL {X  -159.990, Y  +401.273, Z    +0.000, E1   -14.176, E3 +338160.415}
SPL {X  -159.990, Y  +411.788, Z    +0.000, E1   -23.693, E3 +338165.958}
SPL {X  -159.990, Y  +438.158, Z    +0.000, E1   -37.630, E3 +338189.236}
SPL {X  -159.990, Y  +469.969, Z    +0.000, E1   -41.961, E3 +338241.837}
SPL {X  -159.990, Y  +477.498, Z    +0.000, E1   -41.916, E3 +338259.720}
SPL {X  -159.990, Y  +483.140, Z    +0.000, E1   -41.902, E3 +338273.076}
SPL {X  -159.990, Y  +488.618, Z    +0.000, E1   -41.913, E3 +338286.008}
SPL {X  -159.990, Y  +494.299, Z    +0.000, E1   -41.910, E3 +338299.442}
SPL {X  -159.990, Y  +499.538, Z    +0.000, E1   -41.904, E3 +338311.836}
SPL {X  -159.990, Y  +505.259, Z    +0.000, E1   -41.922, E3 +338325.336}
SPL {X  -159.990, Y  +511.862, Z    +0.000, E1   -41.927, E3 +338340.946}
SPL {X  -159.990, Y  +519.146, Z    +0.000, E1   -41.942, E3 +338358.140}
SPL {X  -159.990, Y  +526.974, Z    +0.000, E1   -41.950, E3 +338376.639}
SPL {X  -159.990, Y  +533.758, Z    +0.000, E1   -41.910, E3 +338392.742}
SPL {X  -159.990, Y  +539.474, Z    +0.000, E1   -41.912, E3 +338406.269}
SPL {X  -159.990, Y  +544.879, Z    +0.000, E1   -41.899, E3 +338419.081}
SPL {X  -159.990, Y  +550.802, Z    +0.000, E1   -41.920, E3 +338433.062}
SPL {X  -159.990, Y  +556.952, Z    +0.000, E1   -41.911, E3 +338447.601}
SPL {X  -159.990, Y  +562.629, Z    +0.000, E1   -41.910, E3 +338461.019}
SPL {X  -159.990, Y  +569.054, Z    +0.000, E1   -41.933, E3 +338476.174}
SPL {X  -159.990, Y  +575.562, Z    +0.000, E1   -41.916, E3 +338491.587}
SPL {X  -159.990, Y  +580.118, Z    +0.000, E1   -41.891, E3 +338502.400}
SPL {X  -159.990, Y  +584.320, Z    +0.000, E1   -41.901, E3 +338512.336}
SPL {X  -159.990, Y  +589.217, Z    +0.000, E1   -41.901, E3 +338523.909}
SPL {X  -159.990, Y  +594.252, Z    +0.000, E1   -41.903, E3 +338535.824}
SPL {X  -159.990, Y  +598.793, Z    +0.000, E1   -41.896, E3 +338546.578}
SPL {X  -159.990, Y  +604.215, Z    +0.000, E1   -41.919, E3 +338559.358}
SPL {X  -159.990, Y  +610.545, Z    +0.000, E1   -41.917, E3 +338574.328}
SPL {X  -159.990, Y  +615.720, Z    +0.000, E1   -41.899, E3 +338586.588}
SPL {X  -159.990, Y  +620.005, Z    +0.000, E1   -41.900, E3 +338596.721}
SPL {X  -159.990, Y  +624.919, Z    +0.000, E1   -41.912, E3 +338608.328}
SPL {X  -159.990, Y  +629.282, Z    +0.000, E1   -41.888, E3 +338618.669}
SPL {X  -159.990, Y  +634.411, Z    +0.000, E1   -41.931, E3 +338630.733}
SPL {X  -159.990, Y  +641.479, Z    +0.000, E1   -41.931, E3 +338647.450}
SPL {X  -159.990, Y  +647.782, Z    +0.000, E1   -41.914, E3 +338662.372}
SPL {X  -159.990, Y  +653.094, Z    +0.000, E1   -41.905, E3 +338674.950}
SPL {X  -159.990, Y  +657.893, Z    +0.000, E1   -41.899, E3 +338686.316}
SPL {X  -159.990, Y  +662.516, Z    +0.000, E1   -41.899, E3 +338697.247}
SPL {X  -159.990, Y  +666.974, Z    +0.000, E1   -41.897, E3 +338707.791}
SPL {X  -159.984, Y  +672.859, Z    +0.000, E1   -41.934, E3 +338721.653}
SPL {X  -159.817, Y  +678.937, Z    +0.000, E1   -41.879, E3 +338736.241}
SPL {X  -159.484, Y  +684.213, Z    +0.000, E1   -41.818, E3 +338749.077}
SPL {X  -159.007, Y  +689.209, Z    +0.000, E1   -41.732, E3 +338761.382}
SPL {X  -158.485, Y  +693.390, Z    +0.000, E1   -41.627, E3 +338771.835}
SPL {X  -157.663, Y  +698.690, Z    +0.000, E1   -41.523, E3 +338785.196}
SPL {X  -156.604, Y  +704.242, Z    +0.000, E1   -41.288, E3 +338799.504}
SPL {X  -155.514, Y  +709.078, Z    +0.000, E1   -41.107, E3 +338812.058}
SPL {X  -154.232, Y  +714.035, Z    +0.000, E1   -40.861, E3 +338825.117}
SPL {X  -152.744, Y  +719.104, Z    +0.000, E1   -40.600, E3 +338838.604}
SPL {X  -151.458, Y  +723.048, Z    +0.000, E1   -40.328, E3 +338849.263}
SPL {X  -148.572, Y  +730.857, Z    +0.000, E1   -36.304, E3 +338902.031}
ENDSPLINE

SPLINE
SPL {X  -156.377, Y  +705.307, Z    +0.000, E1   -21.740, E3 +338956.279}
SPL {X  -158.965, Y  +689.585, Z    +0.000, E1   -13.405, E3 +338967.437}
SPL {X  -159.884, Y  +677.314, Z    +0.000, E1    -6.475, E3 +338972.150}
SPL {X  -159.990, Y  +670.142, Z    +0.000, E1    -1.740, E3 +338973.939}
SPL {X  -159.990, Y  +666.629, Z    +0.000, E1    +0.827, E3 +338974.589}
SPL {X  -159.990, Y  +662.407, Z    +0.000, E1    +4.406, E3 +338975.439}
SPL {X  -159.990, Y  +655.884, Z    +0.000, E1   +10.601, E3 +338977.304}
SPL {X  -159.990, Y  +646.242, Z    +0.000, E1   +19.956, E3 +338981.224}
SPL {X  -159.990, Y  +624.365, Z    +0.000, E1   +33.860, E3 +338999.125}
SPL {X  -159.990, Y  +615.596, Z    +0.000, E1   +36.980, E3 +339008.784}
SPL {X  -159.990, Y  +588.349, Z    +0.000, E1   +41.235, E3 +339052.362}
SPL {X  -159.990, Y  +582.302, Z    +0.000, E1   +41.281, E3 +339066.929}
SPL {X  -159.990, Y  +576.269, Z    +0.000, E1   +41.239, E3 +339081.592}
SPL {X  -159.990, Y  +571.714, Z    +0.000, E1   +41.240, E3 +339092.620}
SPL {X  -159.990, Y  +567.050, Z    +0.000, E1   +41.238, E3 +339103.906}
SPL {X  -159.990, Y  +561.959, Z    +0.000, E1   +41.251, E3 +339116.205}
SPL {X  -159.990, Y  +557.719, Z    +0.000, E1   +41.226, E3 +339126.507}
SPL {X  -159.990, Y  +554.148, Z    +0.000, E1   +41.237, E3 +339135.122}
SPL {X  -159.990, Y  +549.897, Z    +0.000, E1   +41.240, E3 +339145.403}
SPL {X  -159.990, Y  +544.775, Z    +0.000, E1   +41.260, E3 +339157.778}
SPL {X  -159.990, Y  +540.176, Z    +0.000, E1   +41.224, E3 +339168.987}
SPL {X  -159.990, Y  +534.009, Z    +0.000, E1   +41.300, E3 +339183.772}
SPL {X  -159.990, Y  +526.579, Z    +0.000, E1   +41.262, E3 +339201.810}
SPL {X  -159.990, Y  +521.454, Z    +0.000, E1   +41.236, E3 +339214.253}
SPL {X  -159.990, Y  +515.605, Z    +0.000, E1   +41.288, E3 +339228.293}
SPL {X  -159.990, Y  +509.898, Z    +0.000, E1   +41.246, E3 +339242.154}
SPL {X  -159.990, Y  +505.215, Z    +0.000, E1   +41.261, E3 +339253.470}
SPL {X  -159.990, Y  +498.837, Z    +0.000, E1   +41.283, E3 +339268.858}
SPL {X  -159.990, Y  +493.848, Z    +0.000, E1   +41.241, E3 +339280.978}
SPL {X  -159.990, Y  +474.734, Z    +0.000, E1   +46.319, E3 +339292.902}
SPL {X  -159.990, Y  +467.791, Z    +0.000, E1   +45.753, E3 +339310.550}
SPL {X  -159.990, Y  +462.409, Z    +0.000, E1   +44.664, E3 +339328.279}
SPL {X  -159.990, Y  +458.229, Z    +0.000, E1   +43.579, E3 +339343.761}
SPL {X  -159.990, Y  +453.434, Z    +0.000, E1   +43.227, E3 +339356.536}
SPL {X  -159.990, Y  +448.702, Z    +0.000, E1   +43.218, E3 +339367.258}
SPL {X  -159.990, Y  +444.476, Z    +0.000, E1   +43.219, E3 +339376.796}
SPL {X  -159.990, Y  +440.246, Z    +0.000, E1   +43.217, E3 +339386.353}
SPL {X  -159.990, Y  +435.724, Z    +0.000, E1   +43.218, E3 +339396.565}
SPL {X  -159.990, Y  +430.527, Z    +0.000, E1   +43.236, E3 +339408.255}
SPL {X  -159.990, Y  +424.433, Z    +0.000, E1   +43.237, E3 +339422.004}
SPL {X  -159.990, Y  +419.466, Z    +0.000, E1   +43.217, E3 +339433.244}
SPL {X  -159.990, Y  +414.585, Z    +0.000, E1   +43.233, E3 +339444.236}
SPL {X  -159.990, Y  +409.927, Z    +0.000, E1   +43.217, E3 +339454.767}
SPL {X  -159.990, Y  +405.428, Z    +0.000, E1   +43.230, E3 +339464.925}
SPL {X  -159.990, Y  +401.033, Z    +0.000, E1   +43.209, E3 +339474.880}
SPL {X  -159.990, Y  +396.968, Z    +0.000, E1   +43.221, E3 +339484.038}
SPL {X  -159.990, Y  +392.163, Z    +0.000, E1   +43.223, E3 +339494.880}
SPL {X  -159.990, Y  +387.342, Z    +0.000, E1   +43.224, E3 +339505.757}
SPL {X  -159.990, Y  +382.548, Z    +0.000, E1   +43.224, E3 +339516.580}
SPL {X  -159.922, Y  +377.835, Z    +0.000, E1   +43.211, E3 +339527.297}
SPL {X  -159.712, Y  +373.072, Z    +0.000, E1   +43.177, E3 +339538.263}
SPL {X  -159.289, Y  +367.537, Z    +0.000, E1   +43.118, E3 +339551.175}
SPL {X  -158.730, Y  +362.464, Z    +0.000, E1   +43.003, E3 +339563.206}
SPL {X  -158.182, Y  +358.518, Z    +0.000, E1   +42.902, E3 +339572.685}
SPL {X  -157.507, Y  +354.423, Z    +0.000, E1   +42.786, E3 +339582.630}
SPL {X  -156.676, Y  +350.104, Z    +0.000, E1   +42.637, E3 +339593.236}
SPL {X  -155.807, Y  +346.154, Z    +0.000, E1   +42.470, E3 +339603.063}
SPL {X  -154.777, Y  +341.993, Z    +0.000, E1   +42.302, E3 +339613.488}
SPL {X  -153.585, Y  +337.686, Z    +0.000, E1   +42.062, E3 +339624.463}
SPL {X  -152.412, Y  +333.846, Z    +0.000, E1   +41.856, E3 +339634.306}
SPL {X  -151.009, Y  +329.651, Z    +0.000, E1   +41.581, E3 +339645.206}
SPL {X  -148.356, Y  +322.607, Z    +0.000, E1   +36.121, E3 +339705.681}
ENDSPLINE

SPLINE
SPL {X  -156.487, Y  +349.204, Z    +0.000, E1   +21.338, E3 +339760.807}
SPL {X  -159.136, Y  +365.992, Z    +0.000, E1   +12.463, E3 +339771.566}
SPL {X  -159.799, Y  +374.694, Z    +0.000, E1    +7.504, E3 +339774.669}
SPL {X  -159.976, Y  +380.404, Z    +0.000, E1    +3.959, E3 +339776.202}
SPL {X  -159.990, Y  +384.773, Z    +0.000, E1    +1.003, E3 +339777.097}
SPL {X  -159.990, Y  +387.968, Z    +0.000, E1    -1.448, E3 +339777.665}
SPL {X  -159.990, Y  +391.397, Z    +0.000, E1    -4.422, E3 +339778.289}
SPL {X  -159.990, Y  +395.864, Z    +0.000, E1    -8.712, E3 +339779.377}
SPL {X  -159.990, Y  +401.273, Z    +0.000, E1   -14.176, E3 +339781.105}
SPL {X  -159.990, Y  +411.788, Z    +0.000, E1   -23.693, E3 +339786.648}
SPL {X  -159.990, Y  +438.158, Z    +0.000, E1   -37.630, E3 +339809.925}
SPL {X  -159.990, Y  +468.567, Z    +0.000, E1   -41.922, E3 +339859.269}
SPL {X  -159.990, Y  +474.616, Z    +0.000, E1   -41.909, E3 +339873.598}
SPL {X  -159.990, Y  +481.610, Z    +0.000, E1   -41.947, E3 +339890.085}
SPL {X  -159.990, Y  +488.618, Z    +0.000, E1   -41.913, E3 +339906.697}
SPL {X  -159.990, Y  +494.299, Z    +0.000, E1   -41.910, E3 +339920.132}
SPL {X  -159.990, Y  +499.538, Z    +0.000, E1   -41.904, E3 +339932.526}
SPL {X  -159.990, Y  +505.259, Z    +0.000, E1   -41.922, E3 +339946.025}
SPL {X  -159.990, Y  +511.862, Z    +0.000, E1   -41.927, E3 +339961.635}
SPL {X  -159.990, Y  +517.450, Z    +0.000, E1   -41.901, E3 +339974.883}
SPL {X  -159.990, Y  +523.027, Z    +0.000, E1   -41.926, E3 +339988.027}
SPL {X  -159.990, Y  +528.611, Z    +0.000, E1   -41.900, E3 +340001.282}
SPL {X  -159.990, Y  +533.758, Z    +0.000, E1   -41.910, E3 +340013.432}
SPL {X  -159.990, Y  +539.474, Z    +0.000, E1   -41.912, E3 +340026.959}
SPL {X  -159.990, Y  +544.879, Z    +0.000, E1   -41.899, E3 +340039.771}
SPL {X  -159.990, Y  +550.802, Z    +0.000, E1   -41.920, E3 +340053.752}
SPL {X  -159.990, Y  +556.952, Z    +0.000, E1   -41.911, E3 +340068.291}
SPL {X  -159.990, Y  +562.629, Z    +0.000, E1   -41.910, E3 +340081.709}
SPL {X  -159.990, Y  +567.682, Z    +0.000, E1   -41.901, E3 +340093.668}
SPL {X  -159.990, Y  +572.912, Z    +0.000, E1   -41.914, E3 +340106.015}
SPL {X  -159.990, Y  +578.863, Z    +0.000, E1   -41.918, E3 +340120.079}
SPL {X  -159.990, Y  +584.320, Z    +0.000, E1   -41.901, E3 +340133.026}
SPL {X  -159.990, Y  +589.217, Z    +0.000, E1   -41.901, E3 +340144.599}
SPL {X  -159.990, Y  +594.252, Z    +0.000, E1   -41.903, E3 +340156.513}
SPL {X  -159.990, Y  +598.793, Z    +0.000, E1   -41.896, E3 +340167.267}
SPL {X  -159.990, Y  +604.215, Z    +0.000, E1   -41.919, E3 +340180.048}
SPL {X  -159.990, Y  +610.545, Z    +0.000, E1   -41.917, E3 +340195.017}
SPL {X  -159.990, Y  +615.720, Z    +0.000, E1   -41.899, E3 +340207.277}
SPL {X  -159.990, Y  +621.417, Z    +0.000, E1   -41.931, E3 +340220.714}
SPL {X  -159.990, Y  +627.900, Z    +0.000, E1   -41.914, E3 +340236.054}
SPL {X  -159.990, Y  +634.411, Z    +0.000, E1   -41.931, E3 +340251.423}
SPL {X  -159.990, Y  +641.479, Z    +0.000, E1   -41.931, E3 +340268.140}
SPL {X  -159.990, Y  +647.782, Z    +0.000, E1   -41.914, E3 +340283.061}
SPL {X  -159.990, Y  +653.094, Z    +0.000, E1   -41.905, E3 +340295.640}
SPL {X  -159.990, Y  +657.893, Z    +0.000, E1   -41.899, E3 +340307.005}
SPL {X  -159.990, Y  +662.516, Z    +0.000, E1   -41.899, E3 +340317.937}
SPL {X  -159.990, Y  +668.411, Z    +0.000, E1   -41.929, E3 +340331.830}
SPL {X  -159.968, Y  +674.139, Z    +0.000, E1   -41.898, E3 +340345.434}
SPL {X  -159.817, Y  +678.937, Z    +0.000, E1   -41.879, E3 +340356.930}
SPL {X  -159.484, Y  +684.213, Z    +0.000, E1   -41.818, E3 +340369.767}
SPL {X  -159.007, Y  +689.209, Z    +0.000, E1   -41.732, E3 +340382.072}
SPL {X  -158.327, Y  +694.511, Z    +0.000, E1   -41.622, E3 +340395.322}
SPL {X  -157.480, Y  +699.729, Z    +0.000, E1   -41.453, E3 +340408.585}
SPL {X  -156.604, Y  +704.242, Z    +0.000, E1   -41.288, E3 +340420.194}
SPL {X  -155.831, Y  +707.744, Z    +0.000, E1   -41.132, E3 +340429.314}
SPL {X  -155.167, Y  +710.488, Z    +0.000, E1   -41.008, E3 +340436.492}
SPL {X  -154.232, Y  +714.035, Z    +0.000, E1   -40.861, E3 +340445.807}
SPL {X  -153.147, Y  +717.790, Z    +0.000, E1   -40.640, E3 +340455.825}
SPL {X  -151.881, Y  +721.788, Z    +0.000, E1   -40.435, E3 +340466.511}
SPL {X  -148.572, Y  +730.857, Z    +0.000, E1   -36.304, E3 +340522.720}
ENDSPLINE

SPLINE
SPL {X  -156.377, Y  +705.307, Z    +0.000, E1   -21.740, E3 +340576.969}
SPL {X  -159.301, Y  +686.331, Z    +0.000, E1   -11.648, E3 +340589.614}
SPL {X  -159.936, Y  +675.651, Z    +0.000, E1    -5.377, E3 +340593.329}
SPL {X  -159.990, Y  +670.142, Z    +0.000, E1    -1.740, E3 +340594.629}
SPL {X  -159.990, Y  +666.629, Z    +0.000, E1    +0.827, E3 +340595.278}
SPL {X  -159.990, Y  +662.407, Z    +0.000, E1    +4.406, E3 +340596.129}
SPL {X  -159.990, Y  +655.884, Z    +0.000, E1   +10.601, E3 +340597.994}
SPL {X  -159.990, Y  +646.242, Z    +0.000, E1   +19.956, E3 +340601.913}
SPL {X  -159.990, Y  +624.365, Z    +0.000, E1   +33.860, E3 +340619.815}
SPL {X  -159.990, Y  +615.596, Z    +0.000, E1   +36.980, E3 +340629.473}
SPL {X  -159.990, Y  +586.905, Z    +0.000, E1   +41.264, E3 +340676.500}
SPL {X  -159.990, Y  +581.111, Z    +0.000, E1   +41.245, E3 +340690.554}
SPL {X  -159.990, Y  +576.269, Z    +0.000, E1   +41.239, E3 +340702.281}
SPL {X  -159.990, Y  +571.714, Z    +0.000, E1   +41.240, E3 +340713.309}
SPL {X  -159.990, Y  +567.050, Z    +0.000, E1   +41.238, E3 +340724.596}
SPL {X  -159.990, Y  +561.959, Z    +0.000, E1   +41.251, E3 +340736.894}
SPL {X  -159.990, Y  +555.553, Z    +0.000, E1   +41.273, E3 +340752.363}
SPL {X  -159.990, Y  +549.897, Z    +0.000, E1   +41.240, E3 +340766.093}
SPL {X  -159.990, Y  +544.775, Z    +0.000, E1   +41.260, E3 +340778.468}
SPL {X  -159.990, Y  +538.952, Z    +0.000, E1   +41.247, E3 +340792.599}
SPL {X  -159.990, Y  +534.225, Z    +0.000, E1   +41.236, E3 +340804.032}
SPL {X  -159.990, Y  +529.136, Z    +0.000, E1   +41.262, E3 +340816.308}
SPL {X  -159.990, Y  +524.776, Z    +0.000, E1   +41.225, E3 +340826.921}
SPL {X  -159.990, Y  +521.454, Z    +0.000, E1   +41.236, E3 +340834.943}
SPL {X  -159.990, Y  +515.605, Z    +0.000, E1   +41.288, E3 +340848.982}
SPL {X  -159.990, Y  +509.898, Z    +0.000, E1   +41.246, E3 +340862.843}
SPL {X  -159.990, Y  +505.215, Z    +0.000, E1   +41.261, E3 +340874.159}
SPL {X  -159.990, Y  +500.102, Z    +0.000, E1   +41.251, E3 +340886.543}
SPL {X  -159.990, Y  +495.023, Z    +0.000, E1   +41.263, E3 +340898.792}
SPL {X  -159.990, Y  +479.011, Z    +0.000, E1   +45.740, E3 +340908.174}
SPL {X  -159.990, Y  +471.379, Z    +0.000, E1   +46.435, E3 +340919.789}
SPL {X  -159.990, Y  +466.895, Z    +0.000, E1   +45.533, E3 +340934.194}
SPL {X  -159.990, Y  +462.409, Z    +0.000, E1   +44.664, E3 +340948.969}
SPL {X  -159.990, Y  +458.229, Z    +0.000, E1   +43.579, E3 +340964.451}
SPL {X  -159.990, Y  +453.434, Z    +0.000, E1   +43.227, E3 +340977.225}
SPL {X  -159.990, Y  +448.702, Z    +0.000, E1   +43.218, E3 +340987.947}
SPL {X  -159.990, Y  +444.476, Z    +0.000, E1   +43.219, E3 +340997.485}
SPL {X  -159.990, Y  +440.246, Z    +0.000, E1   +43.217, E3 +341007.043}
SPL {X  -159.990, Y  +434.411, Z    +0.000, E1   +43.246, E3 +341020.173}
SPL {X  -159.990, Y  +429.216, Z    +0.000, E1   +43.210, E3 +341031.946}
SPL {X  -159.990, Y  +424.433, Z    +0.000, E1   +43.237, E3 +341042.694}
SPL {X  -159.990, Y  +419.466, Z    +0.000, E1   +43.217, E3 +341053.933}
SPL {X  -159.990, Y  +414.585, Z    +0.000, E1   +43.233, E3 +341064.925}
SPL {X  -159.990, Y  +409.927, Z    +0.000, E1   +43.217, E3 +341075.457}
SPL {X  -159.990, Y  +405.428, Z    +0.000, E1   +43.230, E3 +341085.615}
SPL {X  -159.990, Y  +401.033, Z    +0.000, E1   +43.209, E3 +341095.570}
SPL {X  -159.990, Y  +396.968, Z    +0.000, E1   +43.221, E3 +341104.727}
SPL {X  -159.990, Y  +392.163, Z    +0.000, E1   +43.223, E3 +341115.569}
SPL {X  -159.990, Y  +387.342, Z    +0.000, E1   +43.224, E3 +341126.447}
SPL {X  -159.990, Y  +382.548, Z    +0.000, E1   +43.224, E3 +341137.270}
SPL {X  -159.922, Y  +377.835, Z    +0.000, E1   +43.211, E3 +341147.986}
SPL {X  -159.712, Y  +373.072, Z    +0.000, E1   +43.177, E3 +341158.952}
SPL {X  -159.289, Y  +367.537, Z    +0.000, E1   +43.118, E3 +341171.864}
SPL {X  -158.730, Y  +362.464, Z    +0.000, E1   +43.003, E3 +341183.896}
SPL {X  -158.182, Y  +358.518, Z    +0.000, E1   +42.902, E3 +341193.375}
SPL {X  -157.507, Y  +354.423, Z    +0.000, E1   +42.786, E3 +341203.320}
SPL {X  -156.676, Y  +350.104, Z    +0.000, E1   +42.637, E3 +341213.925}
SPL {X  -155.807, Y  +346.154, Z    +0.000, E1   +42.470, E3 +341223.752}
SPL {X  -154.777, Y  +341.993, Z    +0.000, E1   +42.302, E3 +341234.178}
SPL {X  -153.585, Y  +337.686, Z    +0.000, E1   +42.062, E3 +341245.153}
SPL {X  -152.412, Y  +333.846, Z    +0.000, E1   +41.856, E3 +341254.995}
SPL {X  -151.009, Y  +329.651, Z    +0.000, E1   +41.581, E3 +341265.895}
SPL {X  -148.356, Y  +322.607, Z    +0.000, E1   +36.121, E3 +341326.371}
ENDSPLINE

